Yaskawa INFORM job: DEMO_ROOF_SIDE_0625_3PAINT_34.JBI

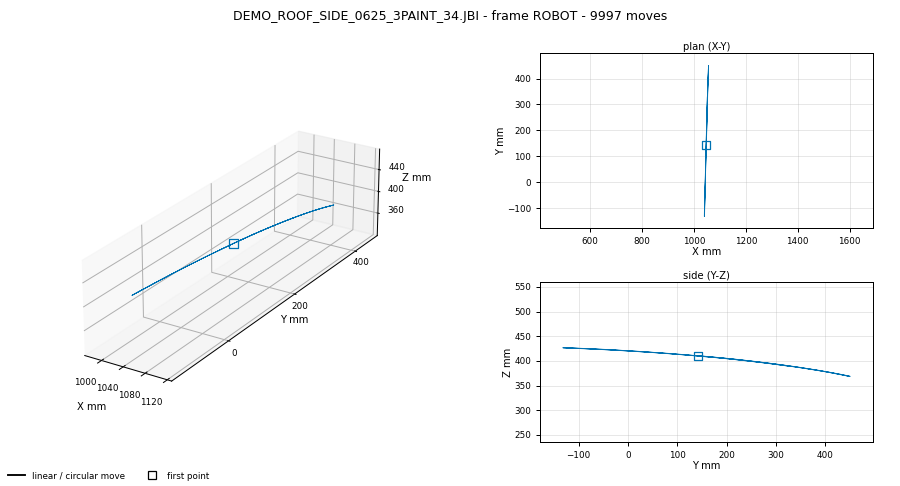
[picture p0: tool path of DEMO_ROOF_SIDE_0625_3PAINT_34.JBI in frame ROBOT, 9997 of 9997 moves have a stored position in this frame; points joined in program order, loops and branches not executed]
/JOB
//NAME DEMO_ROOF_SIDE_0625_3PAINT34
//POS
///NPOS 9997,0,0,0,0,0
///TOOL 0
///USER 0
///POSTYPE ROBOT
///RECTAN
///RCONF 1,0,0,0,0,0,0,0,0,0,0,0,0,0,0,0,0,0,0,0,0,0,0,0
C00000=1047.842,142.026,410.786,170.856,36.125,156.796
C00001=1047.849,142.311,410.761,170.858,36.127,156.797
C00002=1047.855,142.560,410.740,170.860,36.129,156.797
C00003=1047.861,142.809,410.718,170.862,36.131,156.797
C00004=1047.867,143.058,410.697,170.865,36.133,156.798
C00005=1047.873,143.307,410.675,170.866,36.135,156.798
C00006=1047.879,143.556,410.654,170.868,36.136,156.799
C00007=1047.886,143.805,410.633,170.870,36.138,156.799
C00008=1047.892,144.054,410.611,170.872,36.140,156.799
C00009=1047.898,144.303,410.590,170.874,36.142,156.800
C00010=1047.904,144.552,410.568,170.877,36.143,156.800
C00011=1047.910,144.801,410.546,170.878,36.145,156.800
C00012=1047.916,145.050,410.525,170.880,36.147,156.801
C00013=1047.922,145.299,410.504,170.882,36.149,156.801
C00014=1047.928,145.548,410.482,170.884,36.151,156.801
C00015=1047.934,145.797,410.460,170.887,36.153,156.802
C00016=1047.941,146.046,410.438,170.889,36.154,156.802
C00017=1047.947,146.295,410.416,170.890,36.156,156.802
C00018=1047.952,146.544,410.395,170.892,36.158,156.803
C00019=1047.959,146.793,410.373,170.894,36.160,156.803
C00020=1047.965,147.042,410.352,170.897,36.162,156.803
C00021=1047.971,147.291,410.330,170.899,36.164,156.804
C00022=1047.977,147.540,410.308,170.901,36.166,156.804
C00023=1047.983,147.788,410.287,170.903,36.167,156.804
C00024=1047.989,148.038,410.265,170.904,36.169,156.805
C00025=1047.995,148.287,410.243,170.907,36.171,156.805
C00026=1048.001,148.536,410.222,170.909,36.173,156.806
C00027=1048.007,148.785,410.199,170.911,36.175,156.806
C00028=1048.013,149.034,410.177,170.913,36.177,156.806
C00029=1048.019,149.283,410.156,170.915,36.179,156.807
C00030=1048.025,149.532,410.134,170.917,36.180,156.807
C00031=1048.032,149.780,410.112,170.919,36.182,156.807
C00032=1048.038,150.030,410.090,170.921,36.184,156.808
C00033=1048.043,150.279,410.068,170.923,36.186,156.808
C00034=1048.049,150.528,410.046,170.925,36.188,156.808
C00035=1048.055,150.776,410.024,170.927,36.190,156.809
C00036=1048.061,151.025,410.003,170.930,36.192,156.809
C00037=1048.067,151.275,409.981,170.931,36.193,156.809
C00038=1048.073,151.523,409.958,170.933,36.195,156.810
C00039=1048.079,151.773,409.936,170.935,36.197,156.810
C00040=1048.086,152.022,409.915,170.937,36.199,156.811
C00041=1048.092,152.270,409.892,170.940,36.201,156.811
C00042=1048.098,152.519,409.871,170.942,36.203,156.811
C00043=1048.103,152.768,409.848,170.944,36.205,156.812
C00044=1048.109,153.017,409.827,170.946,36.206,156.812
C00045=1048.116,153.266,409.805,170.947,36.208,156.812
C00046=1048.122,153.515,409.783,170.950,36.210,156.813
C00047=1048.128,153.764,409.760,170.952,36.212,156.813
C00048=1048.134,154.013,409.738,170.954,36.214,156.813
C00049=1048.140,154.262,409.716,170.956,36.216,156.814
C00050=1048.147,154.511,409.694,170.958,36.218,156.814
C00051=1048.152,154.760,409.672,170.961,36.219,156.815
C00052=1048.159,155.009,409.649,170.963,36.222,156.815
C00053=1048.164,155.257,409.628,170.965,36.224,156.815
C00054=1048.170,155.506,409.605,170.966,36.226,156.816
C00055=1048.176,155.755,409.584,170.968,36.227,156.816
C00056=1048.182,156.004,409.561,170.971,36.229,156.816
C00057=1048.188,156.254,409.539,170.973,36.231,156.817
C00058=1048.194,156.502,409.517,170.975,36.233,156.817
C00059=1048.201,156.751,409.495,170.977,36.235,156.818
C00060=1048.206,157.000,409.472,170.979,36.237,156.818
C00061=1048.212,157.249,409.450,170.982,36.239,156.818
C00062=1048.219,157.534,409.425,170.984,36.241,156.819
C00063=1048.226,157.820,409.399,170.986,36.244,156.819
C00064=1048.233,158.105,409.373,170.988,36.245,156.820
C00065=1048.240,158.390,409.348,170.991,36.248,156.820
C00066=1048.246,158.639,409.325,170.993,36.250,156.820
C00067=1048.252,158.888,409.304,170.995,36.252,156.821
C00068=1048.258,159.137,409.281,170.997,36.253,156.821
C00069=1048.265,159.386,409.259,170.999,36.255,156.821
C00070=1048.270,159.635,409.236,171.002,36.257,156.822
C00071=1048.277,159.884,409.214,171.004,36.259,156.822
C00072=1048.283,160.132,409.192,171.006,36.261,156.823
C00073=1048.288,160.382,409.169,171.008,36.263,156.823
C00074=1048.295,160.630,409.147,171.011,36.265,156.823
C00075=1048.301,160.879,409.124,171.013,36.267,156.824
C00076=1048.306,161.129,409.102,171.015,36.269,156.824
C00077=1048.312,161.378,409.079,171.017,36.271,156.825
C00078=1048.318,161.626,409.057,171.018,36.273,156.825
C00079=1048.324,161.875,409.034,171.021,36.275,156.825
C00080=1048.330,162.124,409.011,171.023,36.277,156.826
C00081=1048.335,162.373,408.988,171.025,36.279,156.826
C00082=1048.342,162.622,408.966,171.027,36.281,156.827
C00083=1048.347,162.871,408.943,171.030,36.283,156.827
C00084=1048.353,163.120,408.920,171.032,36.285,156.827
C00085=1048.359,163.369,408.897,171.034,36.287,156.828
C00086=1048.365,163.618,408.874,171.036,36.289,156.828
C00087=1048.371,163.866,408.852,171.038,36.292,156.829
C00088=1048.377,164.115,408.829,171.041,36.293,156.829
C00089=1048.382,164.364,408.806,171.043,36.295,156.829
C00090=1048.388,164.614,408.784,171.044,36.298,156.830
C00091=1048.394,164.862,408.761,171.046,36.300,156.830
C00092=1048.400,165.111,408.739,171.049,36.301,156.831
C00093=1048.406,165.360,408.716,171.051,36.304,156.831
C00094=1048.412,165.609,408.693,171.053,36.306,156.831
C00095=1048.417,165.858,408.670,171.055,36.308,156.832
C00096=1048.424,166.106,408.647,171.057,36.310,156.832
C00097=1048.429,166.355,408.624,171.060,36.312,156.833
C00098=1048.435,166.604,408.601,171.062,36.314,156.833
C00099=1048.441,166.853,408.579,171.064,36.316,156.833
C00100=1048.447,167.102,408.556,171.066,36.318,156.834
C00101=1048.452,167.351,408.533,171.069,36.320,156.834
C00102=1048.459,167.599,408.510,171.071,36.322,156.834
C00103=1048.465,167.849,408.487,171.073,36.324,156.835
C00104=1048.471,168.098,408.464,171.075,36.326,156.835
C00105=1048.477,168.347,408.441,171.077,36.328,156.836
C00106=1048.482,168.596,408.418,171.080,36.330,156.836
C00107=1048.489,168.844,408.395,171.082,36.332,156.837
C00108=1048.495,169.093,408.372,171.084,36.334,156.837
C00109=1048.501,169.341,408.349,171.086,36.336,156.837
C00110=1048.506,169.590,408.326,171.089,36.338,156.838
C00111=1048.512,169.839,408.303,171.091,36.340,156.838
C00112=1048.518,170.089,408.280,171.093,36.343,156.839
C00113=1048.525,170.337,408.258,171.095,36.344,156.839
C00114=1048.531,170.586,408.235,171.098,36.346,156.839
C00115=1048.536,170.835,408.212,171.100,36.349,156.840
C00116=1048.542,171.084,408.188,171.102,36.351,156.840
C00117=1048.548,171.332,408.165,171.104,36.352,156.841
C00118=1048.554,171.582,408.142,171.107,36.355,156.841
C00119=1048.561,171.831,408.119,171.109,36.357,156.841
C00120=1048.567,172.080,408.097,171.111,36.358,156.842
C00121=1048.573,172.328,408.073,171.113,36.361,156.842
C00122=1048.578,172.577,408.050,171.115,36.363,156.843
C00123=1048.585,172.826,408.027,171.118,36.365,156.843
C00124=1048.590,173.075,408.004,171.120,36.367,156.843
C00125=1048.596,173.323,407.980,171.122,36.369,156.844
C00126=1048.604,173.609,407.954,171.124,36.371,156.844
C00127=1048.610,173.893,407.928,171.127,36.374,156.845
C00128=1048.618,174.178,407.901,171.130,36.376,156.845
C00129=1048.624,174.463,407.875,171.132,36.378,156.846
C00130=1048.630,174.712,407.852,171.134,36.381,156.846
C00131=1048.636,174.961,407.828,171.137,36.382,156.846
C00132=1048.643,175.209,407.805,171.139,36.384,156.847
C00133=1048.649,175.458,407.782,171.141,36.387,156.847
C00134=1048.655,175.707,407.758,171.143,36.389,156.848
C00135=1048.661,175.956,407.735,171.146,36.390,156.848
C00136=1048.667,176.205,407.712,171.148,36.393,156.849
C00137=1048.673,176.453,407.689,171.150,36.395,156.849
C00138=1048.679,176.703,407.665,171.152,36.397,156.849
C00139=1048.685,176.951,407.642,171.155,36.399,156.850
C00140=1048.691,177.200,407.619,171.158,36.401,156.850
C00141=1048.698,177.449,407.596,171.160,36.403,156.851
C00142=1048.704,177.697,407.572,171.162,36.405,156.851
C00143=1048.710,177.946,407.550,171.164,36.407,156.851
C00144=1048.716,178.195,407.525,171.167,36.409,156.852
C00145=1048.722,178.444,407.503,171.169,36.411,156.852
C00146=1048.728,178.692,407.479,171.171,36.413,156.853
C00147=1048.734,178.942,407.456,171.173,36.415,156.853
C00148=1048.740,179.191,407.433,171.176,36.417,156.853
C00149=1048.746,179.439,407.409,171.178,36.420,156.854
C00150=1048.753,179.689,407.386,171.180,36.422,156.854
C00151=1048.759,179.937,407.362,171.182,36.423,156.855
C00152=1048.765,180.187,407.339,171.186,36.426,156.855
C00153=1048.772,180.435,407.316,171.188,36.428,156.855
C00154=1048.778,180.683,407.292,171.190,36.429,156.856
C00155=1048.784,180.933,407.269,171.192,36.432,156.856
C00156=1048.790,181.181,407.245,171.195,36.434,156.857
C00157=1048.796,181.430,407.222,171.197,36.436,156.857
C00158=1048.802,181.679,407.198,171.199,36.438,156.858
C00159=1048.808,181.928,407.175,171.201,36.440,156.858
C00160=1048.815,182.177,407.151,171.204,36.442,156.858
C00161=1048.821,182.425,407.127,171.207,36.444,156.859
C00162=1048.827,182.674,407.104,171.209,36.447,156.859
C00163=1048.833,182.923,407.080,171.211,36.448,156.860
C00164=1048.840,183.172,407.057,171.213,36.450,156.860
C00165=1048.846,183.421,407.033,171.216,36.453,156.860
C00166=1048.852,183.670,407.009,171.218,36.454,156.861
C00167=1048.858,183.918,406.986,171.220,36.456,156.861
C00168=1048.865,184.167,406.962,171.222,36.459,156.862
C00169=1048.871,184.416,406.939,171.226,36.461,156.862
C00170=1048.876,184.664,406.915,171.228,36.463,156.863
C00171=1048.882,184.914,406.891,171.230,36.465,156.863
C00172=1048.888,185.163,406.867,171.233,36.468,156.864
C00173=1048.894,185.411,406.843,171.235,36.470,156.864
C00174=1048.900,185.660,406.819,171.237,36.472,156.864
C00175=1048.906,185.908,406.795,171.239,36.475,156.865
C00176=1048.911,186.157,406.771,171.242,36.477,156.865
C00177=1048.917,186.406,406.747,171.244,36.479,156.866
C00178=1048.922,186.655,406.723,171.246,36.481,156.866
C00179=1048.929,186.904,406.699,171.249,36.484,156.867
C00180=1048.934,187.153,406.675,171.252,36.486,156.867
C00181=1048.940,187.401,406.651,171.254,36.488,156.868
C00182=1048.947,187.650,406.627,171.256,36.490,156.868
C00183=1048.952,187.899,406.603,171.259,36.493,156.869
C00184=1048.959,188.148,406.579,171.261,36.495,156.869
C00185=1048.964,188.396,406.555,171.263,36.497,156.869
C00186=1048.971,188.645,406.531,171.265,36.500,156.870
C00187=1048.976,188.894,406.506,171.269,36.501,156.870
C00188=1048.983,189.143,406.482,171.271,36.504,156.871
C00189=1048.988,189.391,406.458,171.273,36.506,156.871
C00190=1048.995,189.676,406.431,171.275,36.509,156.872
C00191=1049.002,189.960,406.403,171.279,36.511,156.872
C00192=1049.009,190.244,406.376,171.281,36.514,156.873
C00193=1049.016,190.529,406.347,171.284,36.517,156.873
C00194=1049.022,190.777,406.323,171.287,36.519,156.874
C00195=1049.028,191.027,406.299,171.289,36.521,156.874
C00196=1049.034,191.275,406.275,171.291,36.523,156.875
C00197=1049.040,191.524,406.250,171.293,36.526,156.875
C00198=1049.046,191.772,406.227,171.296,36.528,156.876
C00199=1049.051,192.022,406.202,171.299,36.531,156.876
C00200=1049.058,192.270,406.178,171.301,36.532,156.877
C00201=1049.063,192.519,406.154,171.304,36.535,156.877
C00202=1049.069,192.768,406.130,171.306,36.537,156.878
C00203=1049.076,193.016,406.105,171.308,36.540,156.878
C00204=1049.082,193.264,406.081,171.311,36.541,156.878
C00205=1049.088,193.514,406.057,171.314,36.544,156.879
C00206=1049.094,193.763,406.033,171.316,36.546,156.879
C00207=1049.100,194.011,406.008,171.318,36.549,156.880
C00208=1049.105,194.261,405.984,171.321,36.551,156.880
C00209=1049.112,194.508,405.959,171.324,36.553,156.881
C00210=1049.118,194.758,405.935,171.326,36.555,156.881
C00211=1049.124,195.007,405.911,171.328,36.558,156.882
C00212=1049.130,195.255,405.886,171.331,36.560,156.882
C00213=1049.137,195.503,405.862,171.333,36.562,156.883
C00214=1049.142,195.752,405.837,171.336,36.564,156.883
C00215=1049.149,196.001,405.813,171.339,36.567,156.884
C00216=1049.154,196.250,405.789,171.341,36.569,156.884
C00217=1049.160,196.498,405.764,171.343,36.572,156.885
C00218=1049.167,196.747,405.740,171.346,36.574,156.885
C00219=1049.173,196.997,405.715,171.349,36.576,156.885
C00220=1049.179,197.244,405.691,171.351,36.578,156.886
C00221=1049.185,197.494,405.666,171.353,36.581,156.886
C00222=1049.191,197.743,405.642,171.357,36.583,156.887
C00223=1049.197,197.990,405.617,171.359,36.585,156.887
C00224=1049.203,198.240,405.593,171.361,36.587,156.888
C00225=1049.210,198.488,405.568,171.363,36.590,156.888
C00226=1049.216,198.737,405.543,171.367,36.592,156.889
C00227=1049.222,198.986,405.519,171.369,36.595,156.889
C00228=1049.228,199.234,405.494,171.371,36.597,156.890
C00229=1049.235,199.483,405.470,171.373,36.599,156.890
C00230=1049.241,199.732,405.445,171.377,36.601,156.891
C00231=1049.246,199.981,405.421,171.379,36.604,156.891
C00232=1049.253,200.229,405.396,171.381,36.606,156.892
C00233=1049.259,200.478,405.371,171.384,36.609,156.892
C00234=1049.266,200.727,405.347,171.387,36.611,156.893
C00235=1049.271,200.975,405.322,171.389,36.613,156.893
C00236=1049.277,201.224,405.298,171.392,36.615,156.893
C00237=1049.284,201.473,405.273,171.395,36.618,156.894
C00238=1049.290,201.721,405.247,171.397,36.620,156.894
C00239=1049.296,201.970,405.223,171.399,36.623,156.895
C00240=1049.302,202.219,405.198,171.402,36.625,156.895
C00241=1049.308,202.468,405.173,171.405,36.627,156.896
C00242=1049.314,202.717,405.148,171.407,36.630,156.896
C00243=1049.320,202.965,405.123,171.410,36.632,156.897
C00244=1049.325,203.214,405.098,171.412,36.635,156.897
C00245=1049.332,203.463,405.073,171.415,36.638,156.898
C00246=1049.339,203.711,405.048,171.418,36.640,156.898
C00247=1049.344,203.960,405.024,171.420,36.642,156.899
C00248=1049.350,204.208,404.999,171.423,36.645,156.899
C00249=1049.356,204.457,404.973,171.426,36.647,156.900
C00250=1049.362,204.706,404.949,171.428,36.650,156.900
C00251=1049.368,204.955,404.923,171.430,36.652,156.901
C00252=1049.374,205.203,404.898,171.433,36.655,156.901
C00253=1049.380,205.452,404.873,171.436,36.657,156.902
C00254=1049.406,206.504,404.768,171.671,36.754,156.922
C00255=1049.413,206.762,404.740,171.673,36.758,156.923
C00256=1049.420,207.019,404.713,171.674,36.761,156.924
C00257=1049.426,207.278,404.686,171.677,36.764,156.925
C00258=1049.433,207.535,404.659,171.678,36.768,156.925
C00259=1049.440,207.783,404.633,171.681,36.771,156.926
C00260=1049.446,208.032,404.606,171.683,36.774,156.927
C00261=1049.452,208.281,404.581,171.685,36.777,156.927
C00262=1049.459,208.529,404.555,171.687,36.781,156.928
C00263=1049.465,208.778,404.528,171.689,36.784,156.929
C00264=1049.472,209.026,404.502,171.691,36.787,156.929
C00265=1049.478,209.275,404.476,171.693,36.791,156.930
C00266=1049.485,209.523,404.450,171.695,36.794,156.931
C00267=1049.491,209.772,404.423,171.697,36.797,156.931
C00268=1049.498,210.020,404.397,171.699,36.800,156.932
C00269=1049.504,210.269,404.370,171.701,36.804,156.933
C00270=1049.511,210.518,404.344,171.703,36.807,156.933
C00271=1049.517,210.766,404.318,171.705,36.810,156.934
C00272=1049.523,211.015,404.292,171.707,36.813,156.935
C00273=1049.530,211.263,404.265,171.709,36.816,156.935
C00274=1049.536,211.511,404.239,171.711,36.820,156.936
C00275=1049.543,211.760,404.212,171.714,36.823,156.937
C00276=1049.549,212.008,404.186,171.715,36.826,156.937
C00277=1049.556,212.258,404.159,171.718,36.829,156.938
C00278=1049.562,212.506,404.133,171.719,36.832,156.939
C00279=1049.568,212.754,404.106,171.721,36.836,156.940
C00280=1049.575,213.003,404.080,171.724,36.839,156.940
C00281=1049.581,213.251,404.053,171.725,36.843,156.941
C00282=1049.588,213.500,404.027,171.728,36.846,156.942
C00283=1049.594,213.748,404.000,171.729,36.849,156.942
C00284=1049.599,213.996,403.974,171.732,36.852,156.943
C00285=1049.606,214.245,403.947,171.734,36.856,156.944
C00286=1049.612,214.494,403.921,171.736,36.859,156.944
C00287=1049.619,214.742,403.894,171.738,36.862,156.945
C00288=1049.625,214.991,403.867,171.740,36.865,156.946
C00289=1049.632,215.239,403.841,171.742,36.868,156.946
C00290=1049.638,215.488,403.814,171.744,36.872,156.947
C00291=1049.645,215.737,403.788,171.747,36.875,156.948
C00292=1049.651,215.985,403.761,171.748,36.878,156.948
C00293=1049.658,216.233,403.734,171.751,36.881,156.949
C00294=1049.664,216.481,403.708,171.753,36.884,156.950
C00295=1049.670,216.730,403.681,171.755,36.888,156.951
C00296=1049.677,216.979,403.655,171.757,36.891,156.951
C00297=1049.683,217.228,403.627,171.759,36.894,156.952
C00298=1049.690,217.476,403.601,171.761,36.898,156.953
C00299=1049.696,217.725,403.574,171.763,36.901,156.953
C00300=1049.702,217.972,403.547,171.766,36.904,156.954
C00301=1049.709,218.221,403.521,171.767,36.907,156.955
C00302=1049.716,218.470,403.494,171.770,36.910,156.955
C00303=1049.722,218.718,403.468,171.772,36.913,156.956
C00304=1049.729,218.967,403.440,171.774,36.917,156.957
C00305=1049.735,219.215,403.413,171.776,36.920,156.957
C00306=1049.742,219.464,403.387,171.778,36.923,156.958
C00307=1049.748,219.712,403.360,171.780,36.926,156.959
C00308=1049.755,219.960,403.333,171.782,36.929,156.959
C00309=1049.761,220.209,403.306,171.785,36.932,156.960
C00310=1049.767,220.458,403.279,171.787,36.936,156.961
C00311=1049.774,220.721,403.251,171.789,36.939,156.961
C00312=1049.781,220.984,403.222,171.791,36.942,156.962
C00313=1049.788,221.248,403.194,171.794,36.946,156.963
C00314=1049.795,221.511,403.165,171.796,36.949,156.963
C00315=1049.801,221.759,403.138,171.799,36.952,156.964
C00316=1049.807,222.008,403.111,171.800,36.955,156.965
C00317=1049.814,222.256,403.083,171.802,36.959,156.966
C00318=1049.820,222.505,403.057,171.805,36.962,156.966
C00319=1049.827,222.753,403.030,171.806,36.966,156.967
C00320=1049.833,223.001,403.003,171.809,36.969,156.968
C00321=1049.839,223.250,402.976,171.811,36.972,156.968
C00322=1049.846,223.499,402.948,171.814,36.975,156.969
C00323=1049.852,223.747,402.921,171.815,36.978,156.970
C00324=1049.858,223.996,402.894,171.818,36.981,156.970
C00325=1049.864,224.244,402.867,171.820,36.985,156.971
C00326=1049.872,224.492,402.840,171.822,36.988,156.972
C00327=1049.878,224.741,402.813,171.824,36.991,156.972
C00328=1049.884,224.989,402.786,171.826,36.994,156.973
C00329=1049.890,225.238,402.759,171.829,36.997,156.974
C00330=1049.897,225.486,402.731,171.831,37.001,156.974
C00331=1049.903,225.734,402.703,171.833,37.004,156.975
C00332=1049.910,225.983,402.676,171.835,37.007,156.976
C00333=1049.916,226.232,402.649,171.838,37.010,156.976
C00334=1049.923,226.480,402.623,171.840,37.013,156.977
C00335=1049.929,226.728,402.595,171.843,37.016,156.978
C00336=1049.936,226.977,402.568,171.844,37.019,156.978
C00337=1049.942,227.226,402.540,171.846,37.023,156.979
C00338=1049.949,227.473,402.513,171.849,37.026,156.980
C00339=1049.955,227.722,402.486,171.851,37.029,156.980
C00340=1049.962,227.971,402.458,171.853,37.032,156.981
C00341=1049.968,228.219,402.431,171.855,37.035,156.982
C00342=1049.974,228.468,402.404,171.858,37.038,156.982
C00343=1049.981,228.716,402.376,171.860,37.042,156.983
C00344=1049.988,228.964,402.349,171.863,37.045,156.984
C00345=1049.994,229.213,402.322,171.865,37.048,156.984
C00346=1050.000,229.461,402.294,171.867,37.051,156.985
C00347=1050.007,229.710,402.266,171.869,37.054,156.986
C00348=1050.013,229.958,402.238,171.871,37.057,156.986
C00349=1050.019,230.206,402.211,171.874,37.061,156.987
C00350=1050.026,230.455,402.184,171.876,37.064,156.988
C00351=1050.032,230.703,402.156,171.878,37.067,156.988
C00352=1050.039,230.952,402.129,171.880,37.070,156.989
C00353=1050.045,231.200,402.101,171.883,37.073,156.990
C00354=1050.052,231.448,402.073,171.885,37.076,156.990
C00355=1050.057,231.697,402.046,171.888,37.080,156.991
C00356=1050.064,231.946,402.018,171.889,37.083,156.992
C00357=1050.070,232.194,401.991,171.892,37.086,156.993
C00358=1050.077,232.442,401.963,171.894,37.089,156.993
C00359=1050.084,232.690,401.935,171.896,37.092,156.994
C00360=1050.090,232.939,401.908,171.899,37.095,156.995
C00361=1050.096,233.188,401.879,171.901,37.099,156.995
C00362=1050.102,233.435,401.852,171.904,37.102,156.996
C00363=1050.109,233.684,401.824,171.905,37.105,156.997
C00364=1050.116,233.932,401.796,171.908,37.108,156.997
C00365=1050.122,234.181,401.768,171.910,37.111,156.998
C00366=1050.128,234.429,401.741,171.913,37.115,156.999
C00367=1050.135,234.685,401.712,171.915,37.118,156.999
C00368=1050.141,234.940,401.683,171.918,37.121,157.000
C00369=1050.148,235.197,401.655,171.920,37.124,157.001
C00370=1050.154,235.452,401.626,171.923,37.128,157.002
C00371=1050.160,235.700,401.598,171.924,37.131,157.002
C00372=1050.167,235.949,401.571,171.927,37.133,157.003
C00373=1050.174,236.197,401.543,171.929,37.137,157.004
C00374=1050.180,236.446,401.515,171.932,37.140,157.004
C00375=1050.186,236.695,401.487,171.934,37.143,157.005
C00376=1050.193,236.942,401.459,171.937,37.146,157.006
C00377=1050.199,237.190,401.430,171.939,37.149,157.006
C00378=1050.205,237.439,401.403,171.941,37.152,157.007
C00379=1050.212,237.687,401.375,171.944,37.155,157.008
C00380=1050.219,237.936,401.347,171.945,37.159,157.008
C00381=1050.225,238.184,401.319,171.948,37.162,157.009
C00382=1050.231,238.433,401.291,171.950,37.165,157.010
C00383=1050.238,238.681,401.263,171.953,37.168,157.010
C00384=1050.244,238.930,401.234,171.955,37.171,157.011
C00385=1050.251,239.178,401.207,171.958,37.174,157.012
C00386=1050.257,239.426,401.179,171.960,37.178,157.012
C00387=1050.263,239.674,401.151,171.963,37.181,157.013
C00388=1050.270,239.922,401.123,171.965,37.184,157.014
C00389=1050.276,240.171,401.094,171.968,37.187,157.015
C00390=1050.283,240.419,401.066,171.970,37.190,157.015
C00391=1050.290,240.667,401.038,171.973,37.193,157.016
C00392=1050.296,240.916,401.010,171.975,37.196,157.016
C00393=1050.302,241.164,400.982,171.977,37.200,157.017
C00394=1050.309,241.413,400.954,171.980,37.203,157.018
C00395=1050.315,241.661,400.925,171.981,37.206,157.018
C00396=1050.322,241.909,400.897,171.984,37.209,157.019
C00397=1050.328,242.158,400.868,171.986,37.212,157.020
C00398=1050.334,242.406,400.840,171.989,37.215,157.021
C00399=1050.341,242.655,400.812,171.991,37.219,157.021
C00400=1050.347,242.903,400.783,171.994,37.221,157.022
C00401=1050.354,243.151,400.756,171.996,37.225,157.023
C00402=1050.360,243.400,400.727,171.999,37.228,157.023
C00403=1050.366,243.648,400.698,172.001,37.231,157.024
C00404=1050.373,243.896,400.670,172.004,37.234,157.025
C00405=1050.379,244.145,400.641,172.006,37.237,157.025
C00406=1050.386,244.393,400.613,172.009,37.240,157.026
C00407=1050.392,244.641,400.585,172.011,37.244,157.027
C00408=1050.398,244.890,400.556,172.014,37.247,157.027
C00409=1050.405,245.138,400.528,172.016,37.250,157.028
C00410=1050.411,245.386,400.499,172.019,37.253,157.029
C00411=1050.418,245.635,400.471,172.021,37.256,157.030
C00412=1050.424,245.883,400.442,172.024,37.260,157.030
C00413=1050.430,246.131,400.413,172.026,37.263,157.031
C00414=1050.436,246.380,400.385,172.029,37.266,157.032
C00415=1050.442,246.628,400.356,172.031,37.269,157.032
C00416=1050.449,246.876,400.328,172.034,37.272,157.033
C00417=1050.455,247.124,400.299,172.036,37.276,157.034
C00418=1050.462,247.372,400.270,172.039,37.279,157.034
C00419=1050.468,247.621,400.241,172.041,37.282,157.035
C00420=1050.474,247.869,400.213,172.044,37.285,157.036
C00421=1050.480,248.117,400.184,172.046,37.288,157.036
C00422=1050.486,248.366,400.154,172.049,37.291,157.037
C00423=1050.493,248.615,400.126,172.051,37.294,157.038
C00424=1050.499,248.865,400.097,172.054,37.298,157.039
C00425=1050.505,249.115,400.069,172.056,37.301,157.039
C00426=1050.512,249.365,400.039,172.059,37.304,157.040
C00427=1050.518,249.613,400.010,172.061,37.307,157.041
C00428=1050.524,249.861,399.981,172.064,37.311,157.042
C00429=1050.531,250.109,399.952,172.066,37.314,157.042
C00430=1050.537,250.358,399.923,172.069,37.317,157.043
C00431=1050.543,250.606,399.895,172.071,37.320,157.044
C00432=1050.549,250.855,399.866,172.074,37.323,157.044
C00433=1050.555,251.103,399.837,172.076,37.327,157.045
C00434=1050.562,251.350,399.808,172.079,37.330,157.046
C00435=1050.569,251.599,399.779,172.081,37.333,157.046
C00436=1050.575,251.847,399.750,172.084,37.336,157.047
C00437=1050.582,252.096,399.721,172.086,37.339,157.048
C00438=1050.588,252.344,399.692,172.089,37.343,157.048
C00439=1050.594,252.592,399.663,172.091,37.345,157.049
C00440=1050.600,252.840,399.634,172.094,37.348,157.050
C00441=1050.606,253.089,399.606,172.097,37.352,157.051
C00442=1050.613,253.338,399.576,172.100,37.355,157.051
C00443=1050.620,253.585,399.548,172.102,37.358,157.052
C00444=1050.626,253.833,399.519,172.105,37.361,157.053
C00445=1050.633,254.082,399.490,172.107,37.364,157.053
C00446=1050.639,254.330,399.461,172.110,37.368,157.054
C00447=1050.646,254.579,399.431,172.112,37.371,157.055
C00448=1050.652,254.827,399.402,172.114,37.374,157.055
C00449=1050.659,255.074,399.372,172.117,37.377,157.056
C00450=1050.665,255.322,399.343,172.120,37.380,157.057
C00451=1050.671,255.570,399.314,172.123,37.383,157.057
C00452=1050.678,255.819,399.285,172.126,37.386,157.058
C00453=1050.684,256.067,399.256,172.128,37.389,157.059
C00454=1050.690,256.316,399.227,172.130,37.392,157.060
C00455=1050.697,256.564,399.198,172.133,37.396,157.060
C00456=1050.704,256.812,399.169,172.136,37.399,157.061
C00457=1050.711,257.060,399.140,172.138,37.402,157.062
C00458=1050.717,257.308,399.110,172.142,37.405,157.062
C00459=1050.724,257.557,399.081,172.144,37.408,157.063
C00460=1050.730,257.805,399.052,172.147,37.412,157.064
C00461=1050.736,258.053,399.023,172.149,37.414,157.064
C00462=1050.743,258.301,398.994,172.152,37.417,157.065
C00463=1050.750,258.549,398.963,172.154,37.421,157.066
C00464=1050.756,258.797,398.934,172.157,37.424,157.067
C00465=1050.762,259.046,398.905,172.160,37.427,157.067
C00466=1050.769,259.294,398.876,172.163,37.430,157.068
C00467=1050.776,259.542,398.846,172.165,37.433,157.069
C00468=1050.782,259.790,398.817,172.168,37.436,157.069
C00469=1050.789,260.039,398.788,172.170,37.440,157.070
C00470=1050.795,260.287,398.759,172.173,37.443,157.071
C00471=1050.802,260.535,398.729,172.176,37.445,157.071
C00472=1050.809,260.783,398.700,172.179,37.449,157.072
C00473=1050.815,261.032,398.671,172.181,37.452,157.073
C00474=1050.822,261.280,398.640,172.184,37.455,157.073
C00475=1050.828,261.528,398.611,172.186,37.458,157.074
C00476=1050.834,261.776,398.582,172.190,37.461,157.075
C00477=1050.842,262.024,398.552,172.192,37.464,157.076
C00478=1050.848,262.272,398.523,172.195,37.467,157.076
C00479=1050.855,262.521,398.493,172.197,37.470,157.077
C00480=1050.861,262.769,398.464,172.201,37.473,157.078
C00481=1050.868,263.018,398.435,172.203,37.477,157.078
C00482=1050.874,263.265,398.404,172.206,37.480,157.079
C00483=1050.880,263.513,398.374,172.208,37.483,157.080
C00484=1050.887,263.762,398.345,172.211,37.486,157.080
C00485=1050.894,264.009,398.315,172.214,37.489,157.081
C00486=1050.899,264.258,398.286,172.217,37.493,157.082
C00487=1050.907,264.506,398.256,172.219,37.495,157.083
C00488=1050.913,264.754,398.227,172.222,37.499,157.083
C00489=1050.919,265.002,398.196,172.224,37.502,157.084
C00490=1050.926,265.250,398.166,172.228,37.505,157.085
C00491=1050.932,265.498,398.137,172.230,37.508,157.085
C00492=1050.938,265.747,398.106,172.233,37.512,157.086
C00493=1050.945,265.994,398.077,172.235,37.515,157.087
C00494=1050.951,266.243,398.047,172.239,37.518,157.088
C00495=1050.958,266.491,398.017,172.242,37.521,157.088
C00496=1050.965,266.739,397.987,172.244,37.525,157.089
C00497=1050.970,266.987,397.957,172.247,37.527,157.090
C00498=1050.978,267.236,397.927,172.250,37.531,157.091
C00499=1050.984,267.483,397.897,172.253,37.534,157.091
C00500=1050.990,267.731,397.867,172.255,37.537,157.092
C00501=1050.997,267.980,397.837,172.258,37.540,157.093
C00502=1051.003,268.228,397.807,172.261,37.544,157.093
C00503=1051.010,268.476,397.777,172.264,37.547,157.094
C00504=1051.016,268.723,397.747,172.266,37.550,157.095
C00505=1051.023,268.972,397.716,172.269,37.553,157.096
C00506=1051.029,269.220,397.687,172.272,37.556,157.096
C00507=1051.035,269.469,397.657,172.275,37.559,157.097
C00508=1051.042,269.716,397.627,172.278,37.563,157.098
C00509=1051.048,269.965,397.596,172.281,37.566,157.098
C00510=1051.055,270.212,397.566,172.284,37.569,157.099
C00511=1051.061,270.461,397.536,172.286,37.572,157.100
C00512=1051.068,270.708,397.506,172.289,37.576,157.101
C00513=1051.074,270.957,397.475,172.292,37.579,157.101
C00514=1051.080,271.205,397.445,172.295,37.582,157.102
C00515=1051.087,271.453,397.415,172.297,37.585,157.103
C00516=1051.094,271.701,397.384,172.301,37.588,157.104
C00517=1051.100,271.949,397.354,172.303,37.591,157.104
C00518=1051.107,272.197,397.324,172.306,37.595,157.105
C00519=1051.113,272.445,397.294,172.309,37.598,157.106
C00520=1051.120,272.693,397.263,172.312,37.601,157.106
C00521=1051.125,272.941,397.233,172.315,37.605,157.107
C00522=1051.133,273.189,397.203,172.318,37.607,157.108
C00523=1051.138,273.437,397.172,172.321,37.611,157.109
C00524=1051.145,273.686,397.142,172.323,37.614,157.109
C00525=1051.152,273.934,397.111,172.327,37.617,157.110
C00526=1051.158,274.181,397.080,172.329,37.621,157.111
C00527=1051.165,274.430,397.050,172.332,37.624,157.112
C00528=1051.171,274.677,397.020,172.335,37.627,157.112
C00529=1051.177,274.926,396.989,172.338,37.630,157.113
C00530=1051.184,275.174,396.959,172.341,37.634,157.114
C00531=1051.190,275.422,396.929,172.344,37.636,157.114
C00532=1051.197,275.670,396.897,172.347,37.640,157.115
C00533=1051.203,275.917,396.867,172.349,37.643,157.116
C00534=1051.209,276.166,396.836,172.353,37.646,157.117
C00535=1051.216,276.418,396.805,172.355,37.650,157.117
C00536=1051.222,276.671,396.774,172.359,37.653,157.118
C00537=1051.229,276.923,396.743,172.361,37.656,157.119
C00538=1051.237,277.176,396.711,172.364,37.659,157.120
C00539=1051.243,277.424,396.681,172.368,37.663,157.121
C00540=1051.249,277.672,396.650,172.370,37.666,157.121
C00541=1051.256,277.920,396.619,172.374,37.669,157.122
C00542=1051.262,278.168,396.589,172.376,37.673,157.123
C00543=1051.269,278.416,396.558,172.379,37.676,157.123
C00544=1051.275,278.664,396.527,172.382,37.679,157.124
C00545=1051.281,278.912,396.497,172.385,37.683,157.125
C00546=1051.288,279.160,396.465,172.389,37.685,157.126
C00547=1051.294,279.408,396.434,172.391,37.689,157.126
C00548=1051.301,279.655,396.404,172.394,37.692,157.127
C00549=1051.308,279.904,396.373,172.397,37.695,157.128
C00550=1051.314,280.152,396.342,172.400,37.699,157.129
C00551=1051.321,280.400,396.311,172.403,37.702,157.130
C00552=1051.327,280.647,396.280,172.406,37.705,157.130
C00553=1051.333,280.896,396.249,172.409,37.708,157.131
C00554=1051.340,281.144,396.218,172.412,37.712,157.132
C00555=1051.346,281.391,396.187,172.415,37.715,157.133
C00556=1051.353,281.640,396.156,172.418,37.718,157.133
C00557=1051.359,281.887,396.125,172.421,37.722,157.134
C00558=1051.366,282.135,396.093,172.424,37.725,157.135
C00559=1051.372,282.383,396.063,172.427,37.729,157.136
C00560=1051.379,282.631,396.031,172.430,37.732,157.136
C00561=1051.384,282.880,396.000,172.433,37.735,157.137
C00562=1051.391,283.128,395.969,172.436,37.738,157.138
C00563=1051.397,283.375,395.938,172.439,37.742,157.139
C00564=1051.404,283.623,395.906,172.442,37.745,157.139
C00565=1051.410,283.871,395.876,172.446,37.748,157.140
C00566=1051.417,284.119,395.844,172.448,37.752,157.141
C00567=1051.424,284.367,395.813,172.452,37.755,157.142
C00568=1051.430,284.615,395.781,172.454,37.758,157.142
C00569=1051.436,284.863,395.751,172.458,37.761,157.143
C00570=1051.443,285.111,395.719,172.461,37.765,157.144
C00571=1051.450,285.359,395.688,172.464,37.768,157.145
C00572=1051.456,285.607,395.657,172.467,37.771,157.145
C00573=1051.463,285.855,395.625,172.470,37.775,157.146
C00574=1051.470,286.103,395.594,172.473,37.778,157.147
C00575=1051.476,286.350,395.563,172.477,37.781,157.148
C00576=1051.482,286.598,395.532,172.479,37.784,157.149
C00577=1051.489,286.846,395.500,172.483,37.788,157.149
C00578=1051.496,287.094,395.469,172.485,37.791,157.150
C00579=1051.503,287.342,395.438,172.489,37.795,157.151
C00580=1051.509,287.590,395.406,172.491,37.798,157.152
C00581=1051.515,287.838,395.374,172.495,37.801,157.152
C00582=1051.522,288.086,395.343,172.498,37.804,157.153
C00583=1051.529,288.334,395.311,172.501,37.808,157.154
C00584=1051.535,288.582,395.280,172.504,37.811,157.155
C00585=1051.541,288.830,395.248,172.507,37.815,157.156
C00586=1051.548,289.077,395.217,172.510,37.818,157.156
C00587=1051.554,289.325,395.185,172.514,37.821,157.157
C00588=1051.561,289.573,395.154,172.516,37.824,157.158
C00589=1051.567,289.821,395.122,172.520,37.828,157.159
C00590=1051.574,290.069,395.090,172.523,37.831,157.159
C00591=1051.581,290.333,395.056,172.526,37.835,157.160
C00592=1051.588,290.597,395.023,172.530,37.838,157.161
C00593=1051.594,290.861,394.989,172.533,37.842,157.162
C00594=1051.602,291.125,394.955,172.536,37.846,157.163
C00595=1051.609,291.373,394.924,172.540,37.849,157.164
C00596=1051.615,291.620,394.891,172.542,37.852,157.164
C00597=1051.622,291.868,394.860,172.546,37.856,157.165
C00598=1051.628,292.116,394.828,172.550,37.859,157.166
C00599=1051.634,292.364,394.796,172.552,37.863,157.167
C00600=1051.641,292.611,394.764,172.556,37.866,157.168
C00601=1051.648,292.860,394.732,172.559,37.870,157.168
C00602=1051.654,293.108,394.700,172.562,37.872,157.169
C00603=1051.661,293.355,394.668,172.566,37.876,157.170
C00604=1051.667,293.603,394.636,172.568,37.879,157.171
C00605=1051.674,293.851,394.605,172.572,37.883,157.171
C00606=1051.681,294.098,394.573,172.575,37.886,157.172
C00607=1051.687,294.347,394.541,172.578,37.890,157.173
C00608=1051.694,294.595,394.509,172.582,37.893,157.174
C00609=1051.700,294.842,394.476,172.584,37.896,157.175
C00610=1051.707,295.090,394.445,172.588,37.900,157.176
C00611=1051.713,295.338,394.412,172.591,37.903,157.176
C00612=1051.720,295.586,394.381,172.594,37.907,157.177
C00613=1051.726,295.833,394.348,172.598,37.910,157.178
C00614=1051.733,296.081,394.317,172.601,37.914,157.179
C00615=1051.739,296.329,394.284,172.604,37.917,157.180
C00616=1051.746,296.577,394.253,172.608,37.920,157.180
C00617=1051.752,296.824,394.220,172.611,37.924,157.181
C00618=1051.758,297.072,394.187,172.614,37.928,157.182
C00619=1051.764,297.320,394.155,172.617,37.931,157.183
C00620=1051.771,297.567,394.123,172.621,37.935,157.184
C00621=1051.778,297.816,394.090,172.624,37.938,157.185
C00622=1051.784,298.064,394.058,172.627,37.942,157.185
C00623=1051.790,298.311,394.025,172.631,37.945,157.186
C00624=1051.797,298.559,393.992,172.634,37.949,157.187
C00625=1051.804,298.807,393.961,172.637,37.952,157.188
C00626=1051.810,299.054,393.928,172.640,37.956,157.189
C00627=1051.816,299.302,393.895,172.643,37.960,157.190
C00628=1051.822,299.550,393.863,172.647,37.963,157.190
C00629=1051.828,299.798,393.831,172.651,37.966,157.191
C00630=1051.835,300.045,393.798,172.653,37.970,157.192
C00631=1051.842,300.293,393.765,172.657,37.973,157.193
C00632=1051.849,300.541,393.733,172.661,37.977,157.194
C00633=1051.855,300.789,393.700,172.664,37.981,157.195
C00634=1051.861,301.036,393.667,172.667,37.984,157.195
C00635=1051.868,301.284,393.636,172.671,37.987,157.196
C00636=1051.874,301.532,393.603,172.674,37.991,157.197
C00637=1051.881,301.780,393.570,172.677,37.995,157.198
C00638=1051.887,302.028,393.537,172.681,37.998,157.199
C00639=1051.894,302.275,393.504,172.684,38.002,157.200
C00640=1051.900,302.523,393.472,172.687,38.005,157.200
C00641=1051.907,302.770,393.439,172.691,38.009,157.201
C00642=1051.914,303.018,393.406,172.694,38.012,157.202
C00643=1051.920,303.266,393.374,172.698,38.016,157.203
C00644=1051.926,303.514,393.341,172.701,38.019,157.204
C00645=1051.933,303.761,393.308,172.704,38.023,157.205
C00646=1051.940,304.009,393.275,172.708,38.027,157.206
C00647=1051.947,304.289,393.238,172.712,38.031,157.206
C00648=1051.955,304.568,393.201,172.715,38.035,157.207
C00649=1051.963,304.849,393.164,172.719,38.039,157.208
C00650=1051.970,305.129,393.127,172.723,38.042,157.209
C00651=1051.976,305.376,393.094,172.727,38.046,157.210
C00652=1051.983,305.624,393.061,172.730,38.050,157.211
C00653=1051.989,305.872,393.028,172.734,38.053,157.212
C00654=1051.996,306.119,392.995,172.737,38.057,157.213
C00655=1052.002,306.367,392.962,172.740,38.061,157.214
C00656=1052.009,306.615,392.929,172.744,38.064,157.214
C00657=1052.016,306.862,392.897,172.748,38.068,157.215
C00658=1052.023,307.110,392.864,172.752,38.071,157.216
C00659=1052.030,307.357,392.830,172.754,38.075,157.217
C00660=1052.036,307.605,392.798,172.758,38.079,157.218
C00661=1052.043,307.853,392.764,172.762,38.082,157.219
C00662=1052.050,308.100,392.731,172.765,38.085,157.220
C00663=1052.056,308.349,392.698,172.769,38.089,157.221
C00664=1052.063,308.596,392.665,172.772,38.093,157.221
C00665=1052.069,308.843,392.632,172.775,38.096,157.222
C00666=1052.077,309.091,392.599,172.779,38.100,157.223
C00667=1052.083,309.339,392.566,172.783,38.104,157.224
C00668=1052.090,309.586,392.533,172.787,38.107,157.225
C00669=1052.097,309.834,392.500,172.790,38.111,157.226
C00670=1052.104,310.082,392.467,172.793,38.114,157.227
C00671=1052.110,310.329,392.433,172.797,38.118,157.228
C00672=1052.117,310.578,392.400,172.800,38.122,157.228
C00673=1052.124,310.825,392.367,172.804,38.125,157.229
C00674=1052.131,311.073,392.334,172.808,38.129,157.230
C00675=1052.137,311.320,392.300,172.812,38.132,157.231
C00676=1052.144,311.568,392.267,172.815,38.136,157.232
C00677=1052.151,311.816,392.233,172.819,38.140,157.233
C00678=1052.158,312.063,392.200,172.822,38.143,157.234
C00679=1052.165,312.311,392.167,172.825,38.147,157.234
C00680=1052.171,312.559,392.134,172.829,38.150,157.235
C00681=1052.179,312.806,392.101,172.833,38.154,157.236
C00682=1052.186,313.054,392.067,172.837,38.158,157.237
C00683=1052.192,313.302,392.034,172.840,38.162,157.238
C00684=1052.199,313.549,392.000,172.844,38.165,157.239
C00685=1052.205,313.797,391.966,172.848,38.169,157.240
C00686=1052.212,314.044,391.932,172.851,38.173,157.241
C00687=1052.218,314.292,391.898,172.854,38.177,157.242
C00688=1052.225,314.540,391.865,172.858,38.180,157.243
C00689=1052.231,314.787,391.831,172.862,38.184,157.243
C00690=1052.238,315.035,391.797,172.866,38.188,157.244
C00691=1052.244,315.282,391.763,172.869,38.192,157.245
C00692=1052.251,315.530,391.729,172.873,38.196,157.246
C00693=1052.257,315.777,391.695,172.877,38.199,157.247
C00694=1052.264,316.025,391.662,172.880,38.203,157.248
C00695=1052.270,316.273,391.627,172.883,38.207,157.249
C00696=1052.277,316.520,391.594,172.887,38.211,157.250
C00697=1052.283,316.768,391.559,172.891,38.214,157.251
C00698=1052.290,317.015,391.526,172.895,38.218,157.252
C00699=1052.296,317.263,391.492,172.898,38.222,157.253
C00700=1052.304,317.511,391.458,172.902,38.226,157.254
C00701=1052.309,317.758,391.424,172.906,38.230,157.255
C00702=1052.317,318.006,391.390,172.910,38.233,157.255
C00703=1052.324,318.290,391.351,172.914,38.238,157.257
C00704=1052.331,318.574,391.312,172.919,38.242,157.258
C00705=1052.339,318.858,391.273,172.922,38.247,157.259
C00706=1052.347,319.143,391.233,172.926,38.251,157.260
C00707=1052.353,319.390,391.200,172.930,38.255,157.261
C00708=1052.360,319.637,391.164,172.934,38.259,157.262
C00709=1052.367,319.885,391.131,172.938,38.263,157.263
C00710=1052.373,320.132,391.097,172.941,38.267,157.264
C00711=1052.380,320.380,391.063,172.945,38.270,157.265
C00712=1052.387,320.628,391.028,172.949,38.274,157.265
C00713=1052.394,320.876,390.994,172.953,38.278,157.266
C00714=1052.401,321.123,390.959,172.957,38.282,157.267
C00715=1052.407,321.370,390.925,172.960,38.286,157.268
C00716=1052.414,321.618,390.891,172.964,38.290,157.269
C00717=1052.421,321.865,390.856,172.968,38.294,157.270
C00718=1052.428,322.113,390.822,172.972,38.298,157.271
C00719=1052.434,322.361,390.788,172.976,38.302,157.272
C00720=1052.441,322.608,390.755,172.979,38.306,157.273
C00721=1052.448,322.855,390.719,172.983,38.310,157.274
C00722=1052.454,323.103,390.685,172.987,38.314,157.275
C00723=1052.462,323.350,390.650,172.991,38.317,157.276
C00724=1052.468,323.598,390.616,172.995,38.321,157.277
C00725=1052.475,323.846,390.582,172.998,38.325,157.278
C00726=1052.482,324.093,390.547,173.002,38.329,157.279
C00727=1052.489,324.341,390.513,173.006,38.333,157.280
C00728=1052.496,324.588,390.478,173.011,38.337,157.281
C00729=1052.503,324.836,390.444,173.015,38.341,157.282
C00730=1052.509,325.083,390.410,173.019,38.345,157.283
C00731=1052.516,325.331,390.375,173.022,38.349,157.284
C00732=1052.523,325.578,390.340,173.026,38.353,157.285
C00733=1052.530,325.826,390.306,173.030,38.357,157.286
C00734=1052.537,326.073,390.271,173.034,38.360,157.287
C00735=1052.543,326.321,390.237,173.038,38.364,157.288
C00736=1052.551,326.568,390.202,173.041,38.368,157.289
C00737=1052.557,326.815,390.167,173.045,38.372,157.290
C00738=1052.565,327.063,390.133,173.049,38.376,157.291
C00739=1052.571,327.310,390.098,173.054,38.380,157.292
C00740=1052.578,327.558,390.063,173.058,38.384,157.292
C00741=1052.586,327.806,390.029,173.062,38.388,157.294
C00742=1052.593,328.054,389.994,173.065,38.392,157.295
C00743=1052.599,328.301,389.958,173.069,38.396,157.296
C00744=1052.607,328.549,389.925,173.073,38.400,157.296
C00745=1052.613,328.796,389.889,173.077,38.404,157.297
C00746=1052.620,329.043,389.854,173.081,38.408,157.298
C00747=1052.628,329.290,389.820,173.086,38.412,157.300
C00748=1052.634,329.538,389.785,173.089,38.416,157.301
C00749=1052.641,329.786,389.750,173.093,38.420,157.301
C00750=1052.648,330.034,389.715,173.097,38.424,157.302
C00751=1052.655,330.281,389.680,173.101,38.428,157.304
C00752=1052.662,330.529,389.644,173.105,38.432,157.305
C00753=1052.669,330.776,389.609,173.110,38.436,157.305
C00754=1052.675,331.023,389.574,173.114,38.440,157.307
C00755=1052.682,331.271,389.539,173.118,38.444,157.308
C00756=1052.689,331.518,389.504,173.121,38.449,157.309
C00757=1052.696,331.765,389.469,173.125,38.453,157.310
C00758=1052.702,332.013,389.434,173.129,38.457,157.311
C00759=1052.710,332.292,389.394,173.134,38.462,157.312
C00760=1052.718,332.571,389.354,173.139,38.466,157.313
C00761=1052.726,332.850,389.314,173.143,38.471,157.314
C00762=1052.733,333.129,389.275,173.148,38.475,157.315
C00763=1052.741,333.376,389.239,173.152,38.480,157.316
C00764=1052.748,333.623,389.203,173.156,38.484,157.317
C00765=1052.755,333.871,389.168,173.160,38.488,157.319
C00766=1052.761,334.118,389.133,173.165,38.492,157.320
C00767=1052.768,334.366,389.098,173.169,38.497,157.321
C00768=1052.775,334.613,389.061,173.173,38.501,157.322
C00769=1052.782,334.861,389.026,173.176,38.505,157.323
C00770=1052.789,335.108,388.991,173.180,38.509,157.324
C00771=1052.795,335.355,388.956,173.185,38.513,157.325
C00772=1052.803,335.603,388.920,173.189,38.518,157.326
C00773=1052.810,335.850,388.884,173.193,38.522,157.327
C00774=1052.817,336.097,388.849,173.197,38.526,157.328
C00775=1052.824,336.345,388.813,173.202,38.530,157.329
C00776=1052.830,336.593,388.777,173.206,38.535,157.330
C00777=1052.837,336.839,388.741,173.210,38.539,157.331
C00778=1052.844,337.087,388.706,173.214,38.543,157.332
C00779=1052.852,337.334,388.670,173.219,38.547,157.333
C00780=1052.858,337.582,388.634,173.223,38.552,157.335
C00781=1052.865,337.829,388.599,173.227,38.556,157.336
C00782=1052.872,338.077,388.563,173.232,38.560,157.337
C00783=1052.879,338.324,388.527,173.235,38.565,157.338
C00784=1052.886,338.570,388.491,173.239,38.569,157.339
C00785=1052.893,338.819,388.455,173.243,38.573,157.340
C00786=1052.899,339.066,388.419,173.248,38.578,157.341
C00787=1052.906,339.313,388.384,173.252,38.582,157.342
C00788=1052.914,339.560,388.347,173.256,38.586,157.343
C00789=1052.920,339.807,388.311,173.261,38.590,157.344
C00790=1052.927,340.054,388.275,173.265,38.595,157.345
C00791=1052.935,340.302,388.240,173.269,38.599,157.347
C00792=1052.941,340.549,388.203,173.274,38.604,157.348
C00793=1052.949,340.797,388.167,173.278,38.608,157.349
C00794=1052.955,341.044,388.131,173.282,38.613,157.350
C00795=1052.962,341.292,388.095,173.287,38.617,157.351
C00796=1052.969,341.539,388.059,173.291,38.621,157.352
C00797=1052.976,341.786,388.022,173.295,38.626,157.353
C00798=1052.983,342.033,387.987,173.300,38.630,157.354
C00799=1052.991,342.281,387.950,173.304,38.635,157.356
C00800=1052.997,342.528,387.914,173.308,38.639,157.357
C00801=1053.005,342.776,387.878,173.313,38.643,157.358
C00802=1053.011,343.023,387.842,173.317,38.648,157.359
C00803=1053.019,343.270,387.806,173.322,38.652,157.360
C00804=1053.025,343.517,387.769,173.326,38.657,157.361
C00805=1053.033,343.764,387.732,173.330,38.661,157.362
C00806=1053.039,344.011,387.696,173.335,38.666,157.364
C00807=1053.046,344.259,387.659,173.339,38.670,157.365
C00808=1053.053,344.506,387.623,173.344,38.675,157.366
C00809=1053.060,344.753,387.586,173.348,38.679,157.367
C00810=1053.067,345.000,387.551,173.352,38.684,157.368
C00811=1053.074,345.248,387.514,173.357,38.688,157.369
C00812=1053.081,345.495,387.477,173.361,38.693,157.370
C00813=1053.089,345.742,387.440,173.366,38.697,157.372
C00814=1053.096,345.990,387.404,173.370,38.702,157.373
C00815=1053.104,346.264,387.363,173.375,38.707,157.374
C00816=1053.111,346.539,387.323,173.380,38.712,157.375
C00817=1053.119,346.815,387.281,173.385,38.718,157.377
C00818=1053.127,347.089,387.241,173.390,38.723,157.378
C00819=1053.133,347.336,387.204,173.395,38.727,157.379
C00820=1053.141,347.583,387.167,173.399,38.732,157.380
C00821=1053.148,347.831,387.131,173.404,38.736,157.382
C00822=1053.155,348.077,387.093,173.408,38.741,157.383
C00823=1053.162,348.325,387.057,173.413,38.746,157.384
C00824=1053.169,348.572,387.020,173.417,38.750,157.385
C00825=1053.177,348.820,386.983,173.422,38.755,157.386
C00826=1053.183,349.067,386.946,173.426,38.759,157.387
C00827=1053.190,349.314,386.909,173.431,38.764,157.389
C00828=1053.198,349.561,386.873,173.435,38.769,157.390
C00829=1053.204,349.808,386.836,173.440,38.773,157.391
C00830=1053.212,350.055,386.798,173.445,38.778,157.392
C00831=1053.219,350.303,386.761,173.450,38.783,157.394
C00832=1053.227,350.549,386.724,173.454,38.788,157.395
C00833=1053.234,350.797,386.687,173.459,38.792,157.396
C00834=1053.240,351.044,386.650,173.463,38.797,157.397
C00835=1053.247,351.291,386.613,173.468,38.802,157.398
C00836=1053.254,351.538,386.576,173.472,38.806,157.400
C00837=1053.262,351.786,386.538,173.477,38.811,157.401
C00838=1053.269,352.033,386.501,173.481,38.816,157.402
C00839=1053.276,352.279,386.464,173.486,38.821,157.403
C00840=1053.284,352.526,386.427,173.492,38.826,157.405
C00841=1053.290,352.774,386.390,173.496,38.830,157.406
C00842=1053.298,353.021,386.352,173.501,38.835,157.407
C00843=1053.305,353.268,386.315,173.505,38.840,157.408
C00844=1053.312,353.515,386.277,173.510,38.845,157.410
C00845=1053.319,353.762,386.240,173.514,38.850,157.411
C00846=1053.326,354.009,386.203,173.519,38.855,157.412
C00847=1053.333,354.256,386.165,173.524,38.860,157.413
C00848=1053.341,354.503,386.128,173.528,38.864,157.415
C00849=1053.348,354.750,386.090,173.534,38.869,157.416
C00850=1053.355,354.997,386.053,173.538,38.874,157.417
C00851=1053.362,355.244,386.015,173.543,38.879,157.418
C00852=1053.370,355.492,385.978,173.548,38.884,157.420
C00853=1053.377,355.739,385.940,173.552,38.889,157.421
C00854=1053.384,355.986,385.903,173.557,38.894,157.422
C00855=1053.391,356.233,385.864,173.563,38.898,157.424
C00856=1053.398,356.480,385.827,173.567,38.903,157.425
C00857=1053.405,356.727,385.789,173.572,38.909,157.426
C00858=1053.413,356.974,385.751,173.577,38.914,157.428
C00859=1053.420,357.221,385.714,173.581,38.919,157.429
C00860=1053.427,357.468,385.676,173.587,38.924,157.430
C00861=1053.434,357.715,385.639,173.592,38.928,157.431
C00862=1053.442,357.962,385.600,173.596,38.933,157.433
C00863=1053.449,358.209,385.563,173.601,38.938,157.434
C00864=1053.457,358.456,385.525,173.606,38.944,157.435
C00865=1053.463,358.703,385.486,173.610,38.949,157.437
C00866=1053.470,358.950,385.449,173.616,38.953,157.438
C00867=1053.478,359.197,385.411,173.621,38.959,157.439
C00868=1053.485,359.444,385.373,173.625,38.964,157.441
C00869=1053.492,359.691,385.334,173.630,38.969,157.442
C00870=1053.499,359.938,385.297,173.636,38.974,157.443
C00871=1053.508,360.218,385.253,173.641,38.979,157.445
C00872=1053.516,360.498,385.210,173.646,38.985,157.446
C00873=1053.525,360.778,385.166,173.653,38.991,157.448
C00874=1053.533,361.058,385.124,173.658,38.997,157.449
C00875=1053.540,361.305,385.085,173.663,39.002,157.451
C00876=1053.548,361.551,385.047,173.668,39.007,157.452
C00877=1053.555,361.798,385.010,173.673,39.013,157.453
C00878=1053.562,362.045,384.971,173.678,39.017,157.455
C00879=1053.570,362.292,384.932,173.683,39.023,157.456
C00880=1053.577,362.540,384.895,173.688,39.028,157.458
C00881=1053.584,362.786,384.856,173.693,39.033,157.459
C00882=1053.592,363.033,384.818,173.698,39.039,157.460
C00883=1053.600,363.280,384.779,173.703,39.043,157.462
C00884=1053.607,363.527,384.740,173.709,39.049,157.463
C00885=1053.614,363.773,384.702,173.713,39.054,157.465
C00886=1053.621,364.021,384.664,173.718,39.060,157.466
C00887=1053.629,364.268,384.625,173.724,39.065,157.467
C00888=1053.636,364.515,384.586,173.729,39.070,157.469
C00889=1053.642,364.762,384.548,173.734,39.075,157.470
C00890=1053.650,365.008,384.509,173.739,39.081,157.472
C00891=1053.657,365.256,384.470,173.744,39.086,157.473
C00892=1053.665,365.502,384.431,173.749,39.092,157.474
C00893=1053.672,365.749,384.392,173.755,39.097,157.476
C00894=1053.680,365.996,384.354,173.760,39.102,157.477
C00895=1053.687,366.243,384.315,173.765,39.108,157.479
C00896=1053.695,366.489,384.277,173.770,39.113,157.480
C00897=1053.702,366.737,384.237,173.775,39.119,157.482
C00898=1053.709,366.983,384.199,173.780,39.124,157.483
C00899=1053.717,367.229,384.160,173.786,39.129,157.484
C00900=1053.724,367.477,384.120,173.791,39.135,157.486
C00901=1053.732,367.723,384.082,173.796,39.140,157.487
C00902=1053.739,367.971,384.043,173.802,39.146,157.489
C00903=1053.746,368.217,384.003,173.807,39.151,157.490
C00904=1053.754,368.464,383.965,173.812,39.156,157.492
C00905=1053.761,368.711,383.925,173.818,39.162,157.493
C00906=1053.769,368.957,383.887,173.822,39.168,157.495
C00907=1053.776,369.205,383.848,173.828,39.173,157.496
C00908=1053.783,369.451,383.808,173.833,39.178,157.498
C00909=1053.792,369.698,383.770,173.838,39.184,157.499
C00910=1053.799,369.944,383.730,173.844,39.190,157.501
C00911=1053.806,370.192,383.691,173.849,39.195,157.502
C00912=1053.814,370.438,383.652,173.854,39.200,157.504
C00913=1053.821,370.685,383.613,173.860,39.206,157.505
C00914=1053.830,370.932,383.573,173.865,39.212,157.507
C00915=1053.837,371.179,383.535,173.871,39.218,157.508
C00916=1053.844,371.425,383.495,173.876,39.223,157.510
C00917=1053.853,371.672,383.455,173.881,39.228,157.511
C00918=1053.860,371.919,383.416,173.887,39.234,157.513
C00919=1053.867,372.166,383.377,173.892,39.240,157.514
C00920=1053.875,372.412,383.337,173.898,39.246,157.516
C00921=1053.882,372.659,383.297,173.903,39.251,157.517
C00922=1053.889,372.905,383.258,173.909,39.257,157.519
C00923=1053.897,373.152,383.218,173.914,39.263,157.520
C00924=1053.904,373.400,383.178,173.920,39.269,157.522
C00925=1053.912,373.646,383.139,173.925,39.275,157.523
C00926=1053.919,373.893,383.099,173.931,39.280,157.525
C00927=1053.929,374.191,383.051,173.937,39.287,157.527
C00928=1053.938,374.490,383.002,173.944,39.294,157.529
C00929=1053.947,374.788,382.955,173.951,39.301,157.531
C00930=1053.956,375.087,382.906,173.958,39.308,157.533
C00931=1053.964,375.334,382.866,173.963,39.314,157.534
C00932=1053.971,375.581,382.826,173.969,39.320,157.536
C00933=1053.979,375.827,382.787,173.975,39.326,157.537
C00934=1053.987,376.074,382.747,173.980,39.332,157.539
C00935=1053.995,376.321,382.707,173.986,39.338,157.541
C00936=1054.002,376.568,382.667,173.992,39.344,157.542
C00937=1054.010,376.814,382.626,173.998,39.349,157.544
C00938=1054.018,377.060,382.587,174.003,39.355,157.545
C00939=1054.025,377.307,382.547,174.009,39.361,157.547
C00940=1054.033,377.553,382.506,174.014,39.367,157.549
C00941=1054.041,377.800,382.466,174.020,39.373,157.550
C00942=1054.049,378.047,382.427,174.025,39.379,157.552
C00943=1054.057,378.293,382.386,174.032,39.385,157.554
C00944=1054.065,378.540,382.346,174.038,39.391,157.555
C00945=1054.072,378.786,382.306,174.043,39.397,157.557
C00946=1054.080,379.033,382.266,174.049,39.403,157.558
C00947=1054.087,379.280,382.226,174.054,39.409,157.560
C00948=1054.095,379.526,382.185,174.061,39.415,157.562
C00949=1054.102,379.773,382.145,174.066,39.421,157.563
C00950=1054.110,380.019,382.104,174.072,39.427,157.565
C00951=1054.118,380.266,382.063,174.078,39.433,157.567
C00952=1054.126,380.513,382.024,174.084,39.440,157.568
C00953=1054.134,380.759,381.983,174.090,39.446,157.570
C00954=1054.141,381.006,381.942,174.096,39.452,157.572
C00955=1054.150,381.252,381.901,174.101,39.458,157.573
C00956=1054.157,381.499,381.861,174.107,39.464,157.575
C00957=1054.165,381.745,381.820,174.114,39.471,157.577
C00958=1054.173,381.992,381.779,174.119,39.477,157.579
C00959=1054.181,382.238,381.739,174.125,39.483,157.580
C00960=1054.188,382.484,381.697,174.132,39.489,157.582
C00961=1054.196,382.731,381.657,174.137,39.496,157.584
C00962=1054.204,382.977,381.616,174.143,39.502,157.586
C00963=1054.211,383.224,381.575,174.149,39.508,157.587
C00964=1054.219,383.470,381.534,174.155,39.514,157.589
C00965=1054.227,383.716,381.493,174.161,39.521,157.591
C00966=1054.235,383.963,381.452,174.167,39.527,157.593
C00967=1054.243,384.210,381.411,174.173,39.533,157.594
C00968=1054.250,384.456,381.370,174.179,39.540,157.596
C00969=1054.258,384.703,381.330,174.185,39.546,157.598
C00970=1054.266,384.949,381.289,174.192,39.552,157.600
C00971=1054.274,385.195,381.247,174.197,39.559,157.601
C00972=1054.282,385.441,381.206,174.203,39.566,157.603
C00973=1054.290,385.688,381.165,174.210,39.572,157.605
C00974=1054.298,385.935,381.124,174.216,39.578,157.607
C00975=1054.306,386.180,381.083,174.222,39.585,157.609
C00976=1054.314,386.427,381.042,174.228,39.591,157.610
C00977=1054.322,386.674,381.001,174.235,39.598,157.612
C00978=1054.330,386.920,380.959,174.241,39.604,157.614
C00979=1054.338,387.166,380.918,174.246,39.611,157.616
C00980=1054.346,387.412,380.877,174.253,39.618,157.618
C00981=1054.354,387.659,380.835,174.259,39.624,157.619
C00982=1054.362,387.905,380.794,174.266,39.630,157.621
C00983=1054.373,388.236,380.738,174.274,39.639,157.624
C00984=1054.384,388.567,380.682,174.283,39.648,157.626
C00985=1054.394,388.898,380.627,174.291,39.657,157.629
C00986=1054.406,389.229,380.571,174.300,39.666,157.631
C00987=1054.414,389.475,380.529,174.306,39.673,157.633
C00988=1054.422,389.722,380.488,174.312,39.679,157.635
C00989=1054.430,389.968,380.446,174.318,39.686,157.637
C00990=1054.438,390.214,380.404,174.325,39.693,157.639
C00991=1054.447,390.460,380.363,174.331,39.699,157.641
C00992=1054.454,390.706,380.321,174.338,39.706,157.643
C00993=1054.462,390.953,380.278,174.345,39.713,157.644
C00994=1054.471,391.198,380.237,174.351,39.720,157.646
C00995=1054.479,391.445,380.195,174.358,39.727,157.648
C00996=1054.486,391.691,380.153,174.364,39.734,157.650
C00997=1054.495,391.937,380.111,174.371,39.740,157.652
C00998=1054.503,392.183,380.069,174.376,39.747,157.654
C00999=1054.511,392.430,380.027,174.383,39.754,157.656
C01000=1054.519,392.676,379.985,174.390,39.761,157.658
C01001=1054.528,392.922,379.943,174.396,39.768,157.660
C01002=1054.536,393.169,379.901,174.403,39.775,157.662
C01003=1054.543,393.415,379.859,174.409,39.782,157.664
C01004=1054.552,393.661,379.816,174.416,39.789,157.666
C01005=1054.560,393.907,379.774,174.423,39.796,157.668
C01006=1054.568,394.154,379.732,174.429,39.803,157.670
C01007=1054.576,394.400,379.689,174.436,39.810,157.672
C01008=1054.585,394.645,379.647,174.443,39.817,157.674
C01009=1054.593,394.892,379.605,174.449,39.824,157.676
C01010=1054.601,395.138,379.562,174.456,39.831,157.678
C01011=1054.609,395.384,379.520,174.463,39.838,157.680
C01012=1054.617,395.630,379.477,174.470,39.846,157.682
C01013=1054.626,395.877,379.435,174.476,39.852,157.684
C01014=1054.634,396.123,379.392,174.484,39.860,157.686
C01015=1054.642,396.369,379.350,174.491,39.867,157.688
C01016=1054.650,396.615,379.307,174.497,39.874,157.690
C01017=1054.658,396.861,379.264,174.504,39.881,157.692
C01018=1054.667,397.108,379.221,174.511,39.889,157.694
C01019=1054.675,397.354,379.178,174.518,39.896,157.696
C01020=1054.684,397.600,379.135,174.525,39.903,157.698
C01021=1054.692,397.846,379.093,174.531,39.911,157.700
C01022=1054.700,398.092,379.050,174.538,39.918,157.703
C01023=1054.709,398.338,379.007,174.545,39.925,157.705
C01024=1054.717,398.584,378.964,174.553,39.932,157.707
C01025=1054.726,398.830,378.921,174.559,39.940,157.709
C01026=1054.734,399.076,378.878,174.566,39.948,157.711
C01027=1054.743,399.322,378.835,174.573,39.955,157.713
C01028=1054.750,399.568,378.791,174.580,39.962,157.715
C01029=1054.759,399.814,378.748,174.587,39.970,157.717
C01030=1054.767,400.060,378.705,174.595,39.977,157.720
C01031=1054.776,400.306,378.662,174.602,39.985,157.722
C01032=1054.784,400.553,378.619,174.608,39.992,157.724
C01033=1054.793,400.799,378.576,174.615,40.000,157.726
C01034=1054.801,401.045,378.533,174.623,40.007,157.728
C01035=1054.809,401.290,378.489,174.630,40.015,157.731
C01036=1054.818,401.536,378.446,174.637,40.022,157.733
C01037=1054.827,401.783,378.403,174.644,40.030,157.735
C01038=1054.835,402.029,378.359,174.652,40.038,157.737
C01039=1054.849,402.428,378.288,174.663,40.050,157.741
C01040=1054.863,402.827,378.218,174.675,40.062,157.744
C01041=1054.877,403.227,378.147,174.687,40.075,157.748
C01042=1054.890,403.626,378.076,174.699,40.088,157.752
C01043=1054.899,403.873,378.032,174.706,40.096,157.754
C01044=1054.908,404.118,377.988,174.713,40.103,157.756
C01045=1054.916,404.363,377.945,174.721,40.111,157.758
C01046=1054.924,404.610,377.901,174.728,40.119,157.761
C01047=1054.934,404.856,377.857,174.735,40.127,157.763
C01048=1054.942,405.102,377.813,174.744,40.135,157.765
C01049=1054.951,405.348,377.769,174.751,40.143,157.768
C01050=1054.959,405.594,377.725,174.759,40.151,157.770
C01051=1054.968,405.840,377.681,174.766,40.159,157.772
C01052=1054.976,406.086,377.636,174.774,40.167,157.775
C01053=1054.985,406.332,377.593,174.781,40.175,157.777
C01054=1054.993,406.577,377.548,174.788,40.183,157.779
C01055=1055.002,406.824,377.504,174.796,40.191,157.782
C01056=1055.011,407.069,377.460,174.803,40.199,157.784
C01057=1055.019,407.316,377.415,174.812,40.207,157.786
C01058=1055.028,407.561,377.371,174.819,40.215,157.789
C01059=1055.037,407.807,377.327,174.827,40.224,157.791
C01060=1055.045,408.053,377.282,174.835,40.232,157.794
C01061=1055.055,408.299,377.238,174.842,40.240,157.796
C01062=1055.063,408.544,377.193,174.850,40.248,157.799
C01063=1055.071,408.791,377.148,174.858,40.256,157.801
C01064=1055.080,409.036,377.104,174.866,40.264,157.803
C01065=1055.089,409.282,377.059,174.873,40.273,157.806
C01066=1055.098,409.528,377.015,174.882,40.281,157.808
C01067=1055.107,409.773,376.970,174.889,40.290,157.811
C01068=1055.116,410.020,376.925,174.897,40.298,157.813
C01069=1055.125,410.265,376.881,174.905,40.306,157.816
C01070=1055.133,410.511,376.836,174.913,40.314,157.818
C01071=1055.142,410.757,376.791,174.921,40.323,157.821
C01072=1055.152,411.003,376.747,174.930,40.331,157.823
C01073=1055.161,411.249,376.701,174.937,40.340,157.826
C01074=1055.169,411.495,376.657,174.945,40.348,157.828
C01075=1055.178,411.740,376.612,174.953,40.356,157.831
C01076=1055.187,411.986,376.567,174.961,40.365,157.833
C01077=1055.196,412.232,376.521,174.969,40.373,157.836
C01078=1055.205,412.478,376.477,174.978,40.382,157.838
C01079=1055.215,412.724,376.432,174.985,40.391,157.841
C01080=1055.224,412.970,376.386,174.994,40.400,157.844
C01081=1055.232,413.215,376.341,175.002,40.408,157.846
C01082=1055.242,413.460,376.297,175.011,40.416,157.849
C01083=1055.251,413.706,376.251,175.018,40.425,157.851
C01084=1055.260,413.952,376.206,175.027,40.434,157.854
C01085=1055.269,414.198,376.160,175.035,40.443,157.857
C01086=1055.278,414.444,376.115,175.044,40.452,157.859
C01087=1055.287,414.689,376.069,175.052,40.461,157.862
C01088=1055.296,414.935,376.023,175.061,40.469,157.865
C01089=1055.305,415.180,375.978,175.068,40.479,157.867
C01090=1055.314,415.426,375.932,175.077,40.487,157.870
C01091=1055.328,415.816,375.859,175.091,40.502,157.874
C01092=1055.342,416.207,375.787,175.104,40.515,157.878
C01093=1055.356,416.562,375.721,175.117,40.529,157.882
C01094=1055.369,416.916,375.655,175.129,40.541,157.886
C01095=1055.383,417.270,375.589,175.141,40.555,157.890
C01096=1055.396,417.625,375.522,175.155,40.568,157.894
C01097=1055.405,417.871,375.476,175.163,40.577,157.897
C01098=1055.415,418.116,375.430,175.172,40.586,157.900
C01099=1055.424,418.362,375.384,175.181,40.595,157.903
C01100=1055.433,418.608,375.338,175.190,40.604,157.905
C01101=1055.443,418.853,375.292,175.198,40.614,157.908
C01102=1055.452,419.098,375.245,175.207,40.623,157.911
C01103=1055.462,419.344,375.199,175.216,40.632,157.914
C01104=1055.470,419.589,375.152,175.225,40.642,157.917
C01105=1055.480,419.835,375.106,175.234,40.651,157.920
C01106=1055.490,420.080,375.060,175.243,40.660,157.923
C01107=1055.499,420.326,375.013,175.251,40.670,157.925
C01108=1055.507,420.571,374.967,175.261,40.679,157.928
C01109=1055.517,420.817,374.920,175.270,40.688,157.931
C01110=1055.527,421.062,374.874,175.279,40.698,157.934
C01111=1055.536,421.308,374.826,175.288,40.707,157.937
C01112=1055.545,421.553,374.780,175.297,40.717,157.940
C01113=1055.555,421.799,374.734,175.307,40.727,157.943
C01114=1055.564,422.044,374.686,175.316,40.736,157.946
C01115=1055.574,422.290,374.640,175.325,40.746,157.949
C01116=1055.584,422.534,374.593,175.334,40.756,157.952
C01117=1055.593,422.781,374.546,175.344,40.765,157.955
C01118=1055.602,423.025,374.499,175.353,40.775,157.958
C01119=1055.611,423.271,374.452,175.362,40.785,157.961
C01120=1055.622,423.517,374.405,175.372,40.794,157.964
C01121=1055.631,423.761,374.358,175.381,40.804,157.967
C01122=1055.640,424.007,374.311,175.390,40.814,157.970
C01123=1055.651,424.253,374.263,175.401,40.824,157.973
C01124=1055.659,424.498,374.216,175.410,40.834,157.976
C01125=1055.670,424.743,374.169,175.419,40.843,157.979
C01126=1055.680,424.988,374.121,175.429,40.853,157.982
C01127=1055.689,425.234,374.074,175.438,40.863,157.985
C01128=1055.699,425.478,374.027,175.448,40.874,157.989
C01129=1055.708,425.724,373.979,175.458,40.884,157.992
C01130=1055.719,425.969,373.932,175.468,40.894,157.995
C01131=1055.728,426.215,373.884,175.477,40.904,157.998
C01132=1055.738,426.460,373.837,175.487,40.914,158.001
C01133=1055.748,426.706,373.789,175.497,40.924,158.004
C01134=1055.757,426.951,373.740,175.507,40.934,158.007
C01135=1055.767,427.195,373.694,175.517,40.944,158.011
C01136=1055.776,427.441,373.646,175.527,40.954,158.014
C01137=1055.787,427.686,373.598,175.537,40.965,158.017
C01138=1055.796,427.931,373.550,175.546,40.975,158.020
C01139=1055.806,428.176,373.502,175.557,40.985,158.024
C01140=1055.816,428.421,373.454,175.567,40.996,158.027
C01141=1055.826,428.666,373.406,175.577,41.006,158.030
C01142=1055.836,428.912,373.358,175.587,41.016,158.033
C01143=1055.846,429.157,373.310,175.598,41.027,158.037
C01144=1055.856,429.402,373.261,175.607,41.037,158.040
C01145=1055.866,429.647,373.213,175.618,41.048,158.043
C01146=1055.876,429.893,373.165,175.628,41.058,158.047
C01147=1055.886,430.138,373.117,175.639,41.069,158.050
C01148=1055.896,430.383,373.068,175.649,41.080,158.054
C01149=1055.911,430.759,372.993,175.665,41.096,158.059
C01150=1055.926,431.135,372.919,175.681,41.113,158.064
C01151=1055.942,431.512,372.844,175.697,41.129,158.069
C01152=1055.957,431.888,372.769,175.713,41.145,158.075
C01153=1055.967,432.134,372.720,175.724,41.156,158.078
C01154=1055.978,432.378,372.671,175.734,41.167,158.082
C01155=1055.987,432.623,372.623,175.745,41.178,158.085
C01156=1055.998,432.869,372.574,175.756,41.189,158.089
C01157=1056.008,433.113,372.525,175.767,41.200,158.092
C01158=1056.017,433.358,372.476,175.778,41.211,158.096
C01159=1056.028,433.603,372.426,175.789,41.222,158.099
C01160=1056.039,433.847,372.378,175.800,41.233,158.103
C01161=1056.049,434.093,372.329,175.811,41.245,158.107
C01162=1056.059,434.337,372.280,175.822,41.255,158.110
C01163=1056.070,434.582,372.230,175.833,41.267,158.114
C01164=1056.080,434.828,372.181,175.844,41.278,158.117
C01165=1056.090,435.072,372.132,175.854,41.289,158.121
C01166=1056.101,435.317,372.082,175.866,41.300,158.125
C01167=1056.111,435.562,372.033,175.877,41.312,158.128
C01168=1056.122,435.807,371.983,175.888,41.323,158.132
C01169=1056.133,436.052,371.934,175.899,41.334,158.136
C01170=1056.143,436.296,371.885,175.911,41.346,158.139
C01171=1056.153,436.541,371.835,175.923,41.357,158.143
C01172=1056.164,436.786,371.785,175.934,41.369,158.147
C01173=1056.175,437.031,371.735,175.946,41.380,158.151
C01174=1056.186,437.276,371.685,175.957,41.392,158.155
C01175=1056.195,437.520,371.635,175.968,41.403,158.158
C01176=1056.206,437.765,371.585,175.980,41.415,158.162
C01177=1056.217,438.010,371.536,175.991,41.427,158.166
C01178=1056.228,438.254,371.485,176.004,41.439,158.170
C01179=1056.238,438.499,371.435,176.015,41.450,158.174
C01180=1056.248,438.744,371.385,176.027,41.462,158.178
C01181=1056.259,438.989,371.334,176.038,41.474,158.182
C01182=1056.270,439.233,371.284,176.051,41.486,158.186
C01183=1056.281,439.478,371.235,176.062,41.497,158.189
C01184=1056.291,439.723,371.184,176.074,41.510,158.193
C01185=1056.302,439.967,371.133,176.087,41.521,158.197
C01186=1056.313,440.212,371.083,176.098,41.533,158.201
C01187=1056.323,440.456,371.032,176.111,41.545,158.205
C01188=1056.334,440.701,370.982,176.123,41.557,158.209
C01189=1056.345,440.945,370.931,176.135,41.570,158.213
C01190=1056.356,441.189,370.880,176.147,41.582,158.218
C01191=1056.367,441.434,370.829,176.159,41.594,158.222
C01192=1056.378,441.679,370.778,176.172,41.606,158.226
C01193=1056.389,441.924,370.728,176.185,41.618,158.230
C01194=1056.400,442.168,370.677,176.197,41.631,158.234
C01195=1056.410,442.412,370.626,176.210,41.643,158.238
C01196=1056.422,442.657,370.574,176.222,41.656,158.242
C01197=1056.432,442.902,370.524,176.234,41.668,158.246
C01198=1056.444,443.145,370.473,176.247,41.680,158.251
C01199=1056.455,443.390,370.421,176.259,41.693,158.255
C01200=1056.466,443.635,370.370,176.272,41.706,158.259
C01201=1056.477,443.879,370.318,176.285,41.718,158.263
C01202=1056.488,444.123,370.267,176.299,41.731,158.268
C01203=1056.499,444.368,370.215,176.312,41.743,158.272
C01204=1056.511,444.612,370.164,176.324,41.756,158.276
C01205=1056.529,445.010,370.080,176.345,41.777,158.283
C01206=1056.547,445.406,369.996,176.366,41.797,158.290
C01207=1056.565,445.804,369.912,176.388,41.818,158.298
C01208=1056.584,446.202,369.827,176.410,41.840,158.305
C01209=1056.596,446.445,369.776,176.423,41.853,158.309
C01210=1056.607,446.688,369.724,176.436,41.866,158.314
C01211=1056.619,446.932,369.673,176.450,41.879,158.318
C01212=1056.631,447.176,369.622,176.464,41.891,158.323
C01213=1056.645,447.419,369.571,176.477,41.904,158.327
C01214=1056.659,447.663,369.521,176.491,41.915,158.331
C01215=1056.674,447.907,369.471,176.504,41.928,158.336
C01216=1056.690,448.152,369.423,176.519,41.940,158.340
C01217=1056.707,448.396,369.375,176.533,41.952,158.344
C01218=1056.724,448.641,369.328,176.546,41.963,158.348
C01219=1056.742,448.885,369.280,176.560,41.975,158.352
C01220=1056.762,449.130,369.235,176.575,41.986,158.356
C01221=1056.781,449.375,369.189,176.589,41.997,158.360
C01222=1056.802,449.621,369.143,176.603,42.007,158.364
C01223=1056.824,449.866,369.099,176.617,42.018,158.368
C01224=1056.846,450.111,369.055,176.632,42.028,158.372
C01225=1056.521,450.128,368.769,176.629,42.133,158.401
C01226=1056.499,449.883,368.812,176.614,42.123,158.398
C01227=1056.477,449.637,368.857,176.600,42.113,158.394
C01228=1056.457,449.393,368.902,176.586,42.102,158.390
C01229=1056.435,449.147,368.948,176.571,42.091,158.386
C01230=1056.417,448.902,368.994,176.557,42.080,158.382
C01231=1056.398,448.658,369.041,176.543,42.069,158.378
C01232=1056.381,448.413,369.089,176.528,42.057,158.373
C01233=1056.363,448.168,369.137,176.514,42.046,158.369
C01234=1056.348,447.924,369.185,176.501,42.034,158.365
C01235=1056.332,447.680,369.234,176.487,42.022,158.361
C01236=1056.317,447.436,369.284,176.473,42.010,158.357
C01237=1056.305,447.193,369.334,176.460,41.998,158.352
C01238=1056.291,446.948,369.385,176.445,41.985,158.348
C01239=1056.279,446.705,369.436,176.432,41.972,158.343
C01240=1056.268,446.461,369.489,176.419,41.959,158.339
C01241=1056.257,446.218,369.540,176.405,41.946,158.334
C01242=1056.239,445.841,369.621,176.385,41.926,158.327
C01243=1056.221,445.462,369.701,176.364,41.907,158.321
C01244=1056.203,445.083,369.781,176.344,41.886,158.314
C01245=1056.186,444.705,369.860,176.324,41.867,158.307
C01246=1056.175,444.461,369.912,176.310,41.854,158.303
C01247=1056.164,444.216,369.963,176.297,41.841,158.298
C01248=1056.153,443.972,370.015,176.284,41.829,158.294
C01249=1056.141,443.728,370.067,176.271,41.816,158.290
C01250=1056.131,443.483,370.118,176.258,41.804,158.286
C01251=1056.119,443.239,370.170,176.246,41.791,158.281
C01252=1056.108,442.995,370.221,176.233,41.779,158.277
C01253=1056.097,442.750,370.272,176.220,41.767,158.273
C01254=1056.086,442.506,370.324,176.208,41.754,158.269
C01255=1056.075,442.261,370.374,176.195,41.742,158.264
C01256=1056.064,442.016,370.426,176.182,41.730,158.260
C01257=1056.053,441.772,370.476,176.170,41.718,158.256
C01258=1056.042,441.528,370.527,176.157,41.706,158.252
C01259=1056.031,441.283,370.578,176.145,41.693,158.248
C01260=1056.020,441.038,370.629,176.133,41.681,158.244
C01261=1056.010,440.793,370.680,176.120,41.669,158.240
C01262=1055.999,440.549,370.730,176.108,41.657,158.236
C01263=1055.987,440.305,370.781,176.096,41.645,158.232
C01264=1055.977,440.060,370.832,176.084,41.633,158.228
C01265=1055.966,439.816,370.882,176.072,41.621,158.224
C01266=1055.955,439.572,370.933,176.059,41.609,158.220
C01267=1055.945,439.326,370.983,176.048,41.597,158.216
C01268=1055.934,439.082,371.033,176.036,41.586,158.212
C01269=1055.923,438.837,371.083,176.023,41.574,158.208
C01270=1055.912,438.593,371.134,176.012,41.562,158.204
C01271=1055.902,438.348,371.183,176.000,41.550,158.200
C01272=1055.891,438.103,371.234,175.988,41.539,158.196
C01273=1055.880,437.859,371.285,175.976,41.527,158.192
C01274=1055.870,437.614,371.334,175.965,41.515,158.189
C01275=1055.859,437.369,371.384,175.953,41.504,158.185
C01276=1055.849,437.125,371.434,175.942,41.492,158.181
C01277=1055.838,436.880,371.483,175.930,41.481,158.177
C01278=1055.827,436.635,371.533,175.918,41.470,158.174
C01279=1055.816,436.390,371.583,175.907,41.458,158.170
C01280=1055.806,436.145,371.633,175.895,41.447,158.166
C01281=1055.796,435.901,371.682,175.884,41.435,158.162
C01282=1055.785,435.656,371.732,175.873,41.424,158.158
C01283=1055.774,435.411,371.781,175.861,41.413,158.155
C01284=1055.764,435.166,371.831,175.850,41.402,158.151
C01285=1055.754,434.921,371.880,175.839,41.390,158.148
C01286=1055.743,434.676,371.930,175.828,41.379,158.144
C01287=1055.733,434.432,371.979,175.816,41.368,158.140
C01288=1055.723,434.186,372.028,175.805,41.357,158.137
C01289=1055.712,433.942,372.077,175.794,41.346,158.133
C01290=1055.702,433.697,372.127,175.784,41.335,158.129
C01291=1055.692,433.452,372.175,175.773,41.324,158.126
C01292=1055.681,433.207,372.225,175.762,41.313,158.122
C01293=1055.671,432.963,372.274,175.751,41.302,158.119
C01294=1055.661,432.717,372.323,175.740,41.291,158.115
C01295=1055.651,432.472,372.372,175.730,41.280,158.112
C01296=1055.641,432.228,372.421,175.719,41.269,158.108
C01297=1055.631,431.982,372.470,175.707,41.258,158.105
C01298=1055.615,431.604,372.544,175.691,41.242,158.099
C01299=1055.599,431.226,372.620,175.674,41.225,158.094
C01300=1055.584,430.847,372.696,175.658,41.209,158.089
C01301=1055.568,430.468,372.771,175.642,41.192,158.083
C01302=1055.559,430.223,372.820,175.631,41.182,158.080
C01303=1055.549,429.978,372.868,175.622,41.171,158.077
C01304=1055.539,429.733,372.915,175.611,41.161,158.073
C01305=1055.528,429.488,372.964,175.601,41.150,158.070
C01306=1055.519,429.243,373.013,175.590,41.140,158.067
C01307=1055.508,428.998,373.061,175.580,41.130,158.063
C01308=1055.499,428.752,373.109,175.570,41.119,158.060
C01309=1055.489,428.507,373.157,175.560,41.109,158.057
C01310=1055.478,428.263,373.205,175.549,41.098,158.053
C01311=1055.469,428.017,373.253,175.539,41.088,158.050
C01312=1055.459,427.772,373.301,175.529,41.078,158.047
C01313=1055.449,427.527,373.349,175.519,41.068,158.044
C01314=1055.439,427.282,373.397,175.509,41.057,158.040
C01315=1055.429,427.037,373.444,175.499,41.047,158.037
C01316=1055.420,426.791,373.492,175.489,41.037,158.034
C01317=1055.410,426.546,373.541,175.480,41.027,158.031
C01318=1055.400,426.301,373.588,175.469,41.017,158.028
C01319=1055.391,426.056,373.635,175.459,41.007,158.024
C01320=1055.381,425.811,373.682,175.450,40.997,158.021
C01321=1055.371,425.565,373.730,175.440,40.987,158.018
C01322=1055.361,425.320,373.777,175.430,40.977,158.015
C01323=1055.351,425.074,373.825,175.420,40.967,158.012
C01324=1055.341,424.829,373.873,175.411,40.957,158.009
C01325=1055.331,424.583,373.920,175.402,40.947,158.006
C01326=1055.322,424.339,373.967,175.392,40.937,158.002
C01327=1055.312,424.093,374.014,175.382,40.928,157.999
C01328=1055.303,423.848,374.062,175.372,40.918,157.996
C01329=1055.293,423.603,374.108,175.363,40.908,157.993
C01330=1055.283,423.357,374.156,175.353,40.899,157.990
C01331=1055.274,423.112,374.203,175.344,40.888,157.987
C01332=1055.264,422.866,374.250,175.335,40.879,157.984
C01333=1055.254,422.621,374.297,175.325,40.869,157.981
C01334=1055.245,422.376,374.345,175.316,40.860,157.978
C01335=1055.235,422.130,374.391,175.307,40.850,157.975
C01336=1055.226,421.884,374.438,175.297,40.840,157.972
C01337=1055.217,421.640,374.485,175.288,40.831,157.969
C01338=1055.207,421.394,374.531,175.279,40.821,157.966
C01339=1055.198,421.149,374.579,175.270,40.812,157.963
C01340=1055.188,420.903,374.625,175.260,40.803,157.960
C01341=1055.179,420.658,374.671,175.251,40.793,157.958
C01342=1055.170,420.412,374.718,175.242,40.784,157.955
C01343=1055.160,420.167,374.765,175.233,40.774,157.952
C01344=1055.151,419.922,374.811,175.224,40.765,157.949
C01345=1055.142,419.676,374.857,175.214,40.756,157.946
C01346=1055.132,419.430,374.905,175.206,40.746,157.943
C01347=1055.123,419.185,374.951,175.197,40.737,157.940
C01348=1055.113,418.939,374.997,175.188,40.728,157.938
C01349=1055.104,418.693,375.043,175.179,40.719,157.935
C01350=1055.095,418.448,375.089,175.170,40.709,157.932
C01351=1055.085,418.202,375.135,175.162,40.700,157.929
C01352=1055.076,417.957,375.181,175.153,40.692,157.926
C01353=1055.067,417.712,375.227,175.144,40.682,157.923
C01354=1055.053,417.355,375.294,175.131,40.669,157.919
C01355=1055.040,416.998,375.361,175.118,40.656,157.915
C01356=1055.026,416.642,375.427,175.106,40.643,157.911
C01357=1055.013,416.285,375.494,175.093,40.630,157.907
C01358=1055.004,416.040,375.539,175.084,40.621,157.905
C01359=1054.994,415.794,375.586,175.077,40.612,157.902
C01360=1054.985,415.548,375.631,175.068,40.603,157.899
C01361=1054.976,415.302,375.678,175.059,40.594,157.897
C01362=1054.967,415.057,375.723,175.051,40.586,157.894
C01363=1054.958,414.811,375.769,175.042,40.577,157.891
C01364=1054.949,414.565,375.814,175.034,40.568,157.889
C01365=1054.940,414.320,375.860,175.025,40.559,157.886
C01366=1054.930,414.074,375.905,175.017,40.550,157.883
C01367=1054.921,413.828,375.950,175.008,40.542,157.881
C01368=1054.913,413.583,375.995,175.001,40.533,157.878
C01369=1054.904,413.337,376.041,174.992,40.524,157.875
C01370=1054.895,413.092,376.086,174.984,40.515,157.873
C01371=1054.886,412.846,376.132,174.975,40.507,157.870
C01372=1054.876,412.600,376.177,174.967,40.499,157.868
C01373=1054.867,412.354,376.222,174.959,40.490,157.865
C01374=1054.859,412.108,376.267,174.951,40.482,157.863
C01375=1054.849,411.863,376.311,174.942,40.473,157.860
C01376=1054.840,411.617,376.357,174.935,40.465,157.858
C01377=1054.831,411.371,376.402,174.926,40.456,157.855
C01378=1054.823,411.125,376.447,174.918,40.448,157.853
C01379=1054.813,410.880,376.491,174.910,40.439,157.850
C01380=1054.804,410.634,376.537,174.902,40.431,157.847
C01381=1054.795,410.388,376.581,174.894,40.423,157.845
C01382=1054.787,410.143,376.626,174.886,40.414,157.843
C01383=1054.778,409.896,376.671,174.878,40.406,157.840
C01384=1054.768,409.651,376.716,174.870,40.397,157.837
C01385=1054.760,409.405,376.760,174.862,40.389,157.835
C01386=1054.751,409.158,376.805,174.854,40.381,157.833
C01387=1054.742,408.913,376.849,174.846,40.373,157.830
C01388=1054.734,408.667,376.894,174.839,40.364,157.828
C01389=1054.725,408.421,376.938,174.831,40.357,157.825
C01390=1054.716,408.176,376.983,174.823,40.349,157.823
C01391=1054.707,407.929,377.028,174.815,40.340,157.820
C01392=1054.698,407.684,377.071,174.807,40.332,157.818
C01393=1054.690,407.438,377.116,174.800,40.324,157.816
C01394=1054.682,407.192,377.160,174.792,40.316,157.813
C01395=1054.672,406.946,377.205,174.784,40.308,157.811
C01396=1054.664,406.701,377.250,174.776,40.300,157.809
C01397=1054.654,406.454,377.294,174.769,40.292,157.806
C01398=1054.641,406.071,377.363,174.757,40.279,157.802
C01399=1054.628,405.689,377.431,174.745,40.267,157.799
C01400=1054.615,405.306,377.500,174.733,40.254,157.795
C01401=1054.601,404.923,377.569,174.721,40.242,157.791
C01402=1054.593,404.677,377.612,174.714,40.234,157.789
C01403=1054.584,404.430,377.657,174.707,40.226,157.787
C01404=1054.575,404.185,377.700,174.699,40.219,157.785
C01405=1054.568,403.938,377.744,174.692,40.211,157.782
C01406=1054.559,403.708,377.785,174.685,40.204,157.780
C01407=1054.551,403.478,377.826,174.678,40.196,157.778
C01408=1054.544,403.249,377.867,174.671,40.189,157.776
C01409=1054.536,403.019,377.907,174.664,40.182,157.774
C01410=1054.527,402.790,377.948,174.658,40.175,157.772
C01411=1054.519,402.560,377.989,174.651,40.168,157.770
C01412=1054.511,402.330,378.030,174.644,40.161,157.768
C01413=1054.503,402.100,378.071,174.637,40.153,157.766
C01414=1054.494,401.854,378.114,174.630,40.146,157.763
C01415=1054.486,401.608,378.158,174.623,40.138,157.761
C01416=1054.478,401.362,378.201,174.615,40.130,157.759
C01417=1054.469,401.116,378.244,174.608,40.123,157.757
C01418=1054.461,400.870,378.287,174.601,40.115,157.754
C01419=1054.452,400.625,378.331,174.594,40.108,157.752
C01420=1054.444,400.378,378.374,174.586,40.101,157.750
C01421=1054.434,400.132,378.417,174.579,40.093,157.748
C01422=1054.427,399.885,378.461,174.572,40.086,157.746
C01423=1054.418,399.639,378.504,174.566,40.078,157.744
C01424=1054.410,399.393,378.547,174.559,40.071,157.742
C01425=1054.401,399.147,378.590,174.551,40.063,157.739
C01426=1054.393,398.901,378.633,174.544,40.056,157.737
C01427=1054.384,398.655,378.676,174.537,40.049,157.735
C01428=1054.376,398.410,378.719,174.530,40.041,157.733
C01429=1054.368,398.164,378.762,174.524,40.034,157.731
C01430=1054.359,397.918,378.805,174.516,40.027,157.729
C01431=1054.352,397.671,378.848,174.509,40.019,157.727
C01432=1054.343,397.425,378.891,174.502,40.012,157.725
C01433=1054.335,397.179,378.934,174.495,40.005,157.723
C01434=1054.326,396.932,378.977,174.489,39.998,157.721
C01435=1054.318,396.686,379.019,174.482,39.991,157.718
C01436=1054.310,396.440,379.062,174.475,39.983,157.716
C01437=1054.302,396.194,379.105,174.467,39.976,157.714
C01438=1054.293,395.948,379.147,174.461,39.969,157.712
C01439=1054.284,395.702,379.189,174.454,39.962,157.710
C01440=1054.276,395.455,379.232,174.447,39.955,157.708
C01441=1054.268,395.210,379.274,174.440,39.948,157.706
C01442=1054.260,394.963,379.317,174.434,39.941,157.704
C01443=1054.251,394.717,379.360,174.427,39.934,157.702
C01444=1054.244,394.471,379.402,174.420,39.927,157.700
C01445=1054.235,394.225,379.445,174.414,39.919,157.698
C01446=1054.227,393.978,379.487,174.407,39.913,157.696
C01447=1054.219,393.733,379.528,174.400,39.906,157.694
C01448=1054.211,393.486,379.571,174.394,39.898,157.692
C01449=1054.202,393.240,379.614,174.387,39.892,157.690
C01450=1054.195,392.994,379.656,174.380,39.885,157.688
C01451=1054.186,392.747,379.698,174.374,39.878,157.686
C01452=1054.179,392.501,379.740,174.367,39.871,157.684
C01453=1054.170,392.255,379.782,174.361,39.864,157.682
C01454=1054.161,392.009,379.825,174.354,39.857,157.680
C01455=1054.154,391.763,379.867,174.347,39.851,157.678
C01456=1054.145,391.517,379.908,174.341,39.844,157.677
C01457=1054.137,391.271,379.950,174.334,39.837,157.675
C01458=1054.129,391.024,379.993,174.328,39.830,157.673
C01459=1054.121,390.778,380.033,174.321,39.823,157.671
C01460=1054.113,390.531,380.075,174.314,39.816,157.669
C01461=1054.105,390.285,380.117,174.308,39.810,157.667
C01462=1054.097,390.039,380.159,174.302,39.803,157.665
C01463=1054.089,389.793,380.201,174.296,39.796,157.663
C01464=1054.081,389.547,380.243,174.289,39.790,157.661
C01465=1054.072,389.300,380.285,174.283,39.783,157.659
C01466=1054.062,388.967,380.341,174.274,39.774,157.657
C01467=1054.051,388.635,380.397,174.266,39.765,157.654
C01468=1054.039,388.302,380.453,174.257,39.756,157.652
C01469=1054.029,387.970,380.508,174.248,39.747,157.649
C01470=1054.021,387.723,380.550,174.242,39.741,157.648
C01471=1054.013,387.477,380.591,174.236,39.734,157.646
C01472=1054.004,387.230,380.633,174.229,39.728,157.644
C01473=1053.996,386.984,380.674,174.224,39.721,157.642
C01474=1053.988,386.738,380.715,174.217,39.715,157.640
C01475=1053.981,386.492,380.756,174.211,39.708,157.638
C01476=1053.972,386.245,380.798,174.204,39.702,157.637
C01477=1053.964,385.999,380.839,174.198,39.696,157.635
C01478=1053.957,385.752,380.880,174.193,39.689,157.633
C01479=1053.948,385.507,380.921,174.186,39.683,157.631
C01480=1053.940,385.259,380.963,174.180,39.677,157.629
C01481=1053.932,385.013,381.004,174.173,39.670,157.628
C01482=1053.924,384.767,381.044,174.168,39.664,157.626
C01483=1053.917,384.520,381.086,174.162,39.657,157.624
C01484=1053.909,384.274,381.127,174.155,39.651,157.622
C01485=1053.901,384.027,381.168,174.149,39.645,157.621
C01486=1053.893,383.781,381.209,174.144,39.638,157.619
C01487=1053.885,383.535,381.250,174.137,39.632,157.617
C01488=1053.877,383.288,381.291,174.131,39.626,157.615
C01489=1053.869,383.042,381.332,174.125,39.619,157.614
C01490=1053.861,382.795,381.372,174.119,39.613,157.612
C01491=1053.854,382.549,381.413,174.113,39.607,157.610
C01492=1053.846,382.303,381.454,174.107,39.601,157.608
C01493=1053.838,382.056,381.495,174.101,39.594,157.607
C01494=1053.831,381.810,381.536,174.095,39.589,157.605
C01495=1053.823,381.563,381.576,174.089,39.582,157.603
C01496=1053.815,381.317,381.617,174.083,39.576,157.601
C01497=1053.808,381.070,381.658,174.077,39.570,157.600
C01498=1053.800,380.824,381.698,174.071,39.564,157.598
C01499=1053.792,380.577,381.739,174.065,39.557,157.596
C01500=1053.785,380.330,381.780,174.060,39.551,157.595
C01501=1053.777,380.084,381.820,174.054,39.545,157.593
C01502=1053.769,379.838,381.861,174.048,39.539,157.591
C01503=1053.761,379.591,381.901,174.042,39.533,157.590
C01504=1053.753,379.344,381.941,174.036,39.527,157.588
C01505=1053.745,379.097,381.981,174.031,39.521,157.586
C01506=1053.737,378.851,382.022,174.024,39.515,157.585
C01507=1053.729,378.604,382.062,174.019,39.509,157.583
C01508=1053.721,378.358,382.102,174.013,39.503,157.581
C01509=1053.714,378.111,382.142,174.007,39.497,157.580
C01510=1053.706,377.865,382.183,174.002,39.491,157.578
C01511=1053.699,377.619,382.223,173.995,39.485,157.577
C01512=1053.691,377.372,382.262,173.990,39.479,157.575
C01513=1053.683,377.125,382.303,173.984,39.474,157.573
C01514=1053.675,376.879,382.343,173.978,39.468,157.572
C01515=1053.667,376.632,382.383,173.973,39.462,157.570
C01516=1053.660,376.385,382.423,173.967,39.456,157.568
C01517=1053.652,376.139,382.463,173.962,39.450,157.567
C01518=1053.644,375.892,382.503,173.956,39.444,157.565
C01519=1053.637,375.645,382.543,173.950,39.438,157.564
C01520=1053.629,375.398,382.583,173.944,39.432,157.562
C01521=1053.622,375.152,382.622,173.939,39.427,157.560
C01522=1053.612,374.851,382.671,173.932,39.420,157.559
C01523=1053.603,374.551,382.720,173.925,39.413,157.557
C01524=1053.594,374.250,382.768,173.918,39.406,157.555
C01525=1053.584,373.949,382.817,173.911,39.399,157.553
C01526=1053.577,373.703,382.857,173.906,39.393,157.551
C01527=1053.570,373.456,382.897,173.900,39.387,157.550
C01528=1053.562,373.209,382.937,173.895,39.382,157.548
C01529=1053.554,372.963,382.976,173.889,39.376,157.547
C01530=1053.546,372.716,383.015,173.884,39.370,157.545
C01531=1053.540,372.470,383.054,173.878,39.364,157.544
C01532=1053.532,372.223,383.094,173.873,39.359,157.542
C01533=1053.524,371.976,383.134,173.867,39.353,157.540
C01534=1053.517,371.730,383.174,173.862,39.347,157.539
C01535=1053.510,371.482,383.213,173.856,39.342,157.537
C01536=1053.501,371.236,383.252,173.851,39.336,157.536
C01537=1053.494,370.989,383.292,173.846,39.331,157.534
C01538=1053.487,370.742,383.331,173.840,39.325,157.533
C01539=1053.479,370.496,383.370,173.835,39.319,157.531
C01540=1053.471,370.248,383.409,173.829,39.314,157.530
C01541=1053.464,370.002,383.449,173.824,39.309,157.528
C01542=1053.456,369.756,383.488,173.818,39.303,157.527
C01543=1053.448,369.508,383.527,173.813,39.297,157.525
C01544=1053.440,369.262,383.566,173.808,39.292,157.524
C01545=1053.433,369.015,383.605,173.802,39.287,157.522
C01546=1053.426,368.768,383.644,173.797,39.281,157.521
C01547=1053.418,368.521,383.684,173.791,39.275,157.519
C01548=1053.411,368.274,383.722,173.787,39.270,157.518
C01549=1053.403,368.028,383.761,173.782,39.265,157.517
C01550=1053.396,367.781,383.801,173.776,39.259,157.515
C01551=1053.389,367.534,383.839,173.771,39.254,157.514
C01552=1053.381,367.287,383.878,173.765,39.248,157.512
C01553=1053.374,367.041,383.918,173.760,39.243,157.511
C01554=1053.365,366.794,383.956,173.755,39.238,157.509
C01555=1053.359,366.547,383.995,173.749,39.232,157.508
C01556=1053.352,366.300,384.034,173.744,39.227,157.506
C01557=1053.344,366.053,384.072,173.740,39.221,157.505
C01558=1053.337,365.806,384.112,173.734,39.216,157.504
C01559=1053.329,365.560,384.150,173.729,39.211,157.502
C01560=1053.322,365.312,384.189,173.724,39.205,157.501
C01561=1053.314,365.066,384.228,173.718,39.200,157.499
C01562=1053.307,364.819,384.266,173.713,39.195,157.498
C01563=1053.300,364.573,384.305,173.708,39.190,157.496
C01564=1053.292,364.325,384.344,173.703,39.184,157.495
C01565=1053.285,364.078,384.383,173.698,39.179,157.494
C01566=1053.278,363.832,384.421,173.693,39.174,157.492
C01567=1053.271,363.585,384.460,173.687,39.169,157.491
C01568=1053.263,363.338,384.498,173.682,39.163,157.489
C01569=1053.255,363.091,384.537,173.678,39.158,157.488
C01570=1053.249,362.844,384.575,173.672,39.153,157.487
C01571=1053.241,362.597,384.613,173.667,39.147,157.485
C01572=1053.233,362.350,384.652,173.662,39.143,157.484
C01573=1053.226,362.103,384.691,173.657,39.137,157.482
C01574=1053.219,361.856,384.728,173.652,39.132,157.481
C01575=1053.212,361.609,384.766,173.647,39.127,157.480
C01576=1053.204,361.362,384.805,173.642,39.122,157.478
C01577=1053.197,361.115,384.843,173.636,39.117,157.477
C01578=1053.189,360.833,384.887,173.631,39.111,157.476
C01579=1053.180,360.552,384.930,173.626,39.105,157.474
C01580=1053.172,360.270,384.974,173.620,39.099,157.472
C01581=1053.164,359.988,385.018,173.614,39.093,157.471
C01582=1053.156,359.741,385.056,173.610,39.088,157.470
C01583=1053.149,359.494,385.093,173.604,39.084,157.468
C01584=1053.141,359.248,385.132,173.599,39.079,157.467
C01585=1053.134,359.001,385.169,173.594,39.073,157.466
C01586=1053.128,358.753,385.207,173.590,39.068,157.464
C01587=1053.120,358.507,385.245,173.584,39.064,157.463
C01588=1053.113,358.260,385.283,173.579,39.059,157.462
C01589=1053.105,358.012,385.322,173.575,39.053,157.460
C01590=1053.098,357.765,385.360,173.570,39.048,157.459
C01591=1053.091,357.518,385.397,173.565,39.044,157.458
C01592=1053.083,357.271,385.435,173.560,39.039,157.456
C01593=1053.076,357.024,385.473,173.555,39.034,157.455
C01594=1053.069,356.777,385.511,173.550,39.029,157.454
C01595=1053.062,356.530,385.548,173.546,39.024,157.453
C01596=1053.054,356.283,385.586,173.541,39.019,157.451
C01597=1053.047,356.036,385.624,173.535,39.014,157.450
C01598=1053.040,355.789,385.661,173.531,39.009,157.449
C01599=1053.032,355.542,385.699,173.526,39.004,157.447
C01600=1053.025,355.295,385.736,173.521,39.000,157.446
C01601=1053.018,355.048,385.774,173.517,38.995,157.445
C01602=1053.011,354.801,385.811,173.512,38.990,157.444
C01603=1053.003,354.553,385.849,173.507,38.985,157.442
C01604=1052.997,354.307,385.886,173.502,38.980,157.441
C01605=1052.989,354.060,385.924,173.497,38.975,157.440
C01606=1052.982,353.813,385.961,173.493,38.970,157.438
C01607=1052.975,353.566,385.999,173.488,38.966,157.437
C01608=1052.968,353.318,386.036,173.484,38.961,157.436
C01609=1052.960,353.071,386.074,173.478,38.956,157.435
C01610=1052.953,352.824,386.111,173.473,38.951,157.433
C01611=1052.946,352.577,386.149,173.469,38.946,157.432
C01612=1052.940,352.330,386.185,173.464,38.942,157.431
C01613=1052.932,352.083,386.223,173.460,38.937,157.430
C01614=1052.925,351.836,386.260,173.455,38.932,157.428
C01615=1052.918,351.589,386.298,173.451,38.927,157.427
C01616=1052.911,351.341,386.335,173.446,38.923,157.426
C01617=1052.904,351.095,386.371,173.441,38.918,157.425
C01618=1052.896,350.848,386.409,173.436,38.913,157.423
C01619=1052.889,350.600,386.446,173.432,38.908,157.422
C01620=1052.882,350.353,386.483,173.427,38.904,157.421
C01621=1052.875,350.105,386.521,173.422,38.899,157.420
C01622=1052.868,349.859,386.556,173.418,38.894,157.419
C01623=1052.861,349.612,386.594,173.413,38.890,157.417
C01624=1052.854,349.364,386.631,173.409,38.885,157.416
C01625=1052.846,349.117,386.668,173.404,38.881,157.415
C01626=1052.839,348.870,386.704,173.399,38.876,157.414
C01627=1052.832,348.623,386.742,173.394,38.871,157.413
C01628=1052.825,348.375,386.779,173.390,38.866,157.411
C01629=1052.819,348.129,386.816,173.385,38.862,157.410
C01630=1052.811,347.881,386.852,173.381,38.857,157.409
C01631=1052.804,347.634,386.889,173.377,38.853,157.408
C01632=1052.797,347.386,386.926,173.372,38.848,157.407
C01633=1052.790,347.140,386.962,173.368,38.843,157.405
C01634=1052.781,346.863,387.004,173.363,38.838,157.404
C01635=1052.773,346.586,387.045,173.358,38.834,157.403
C01636=1052.766,346.310,387.086,173.352,38.828,157.401
C01637=1052.758,346.033,387.127,173.347,38.823,157.400
C01638=1052.751,345.786,387.164,173.343,38.819,157.399
C01639=1052.744,345.539,387.200,173.338,38.814,157.398
C01640=1052.737,345.291,387.237,173.334,38.809,157.397
C01641=1052.730,345.044,387.273,173.329,38.805,157.396
C01642=1052.723,344.797,387.310,173.325,38.801,157.394
C01643=1052.716,344.549,387.346,173.321,38.796,157.393
C01644=1052.709,344.303,387.384,173.316,38.792,157.392
C01645=1052.701,344.055,387.420,173.312,38.787,157.391
C01646=1052.695,343.808,387.456,173.307,38.783,157.390
C01647=1052.687,343.561,387.492,173.303,38.778,157.389
C01648=1052.681,343.314,387.529,173.299,38.774,157.388
C01649=1052.673,343.066,387.565,173.294,38.769,157.386
C01650=1052.667,342.819,387.601,173.290,38.765,157.385
C01651=1052.659,342.572,387.638,173.286,38.761,157.384
C01652=1052.653,342.325,387.674,173.281,38.756,157.383
C01653=1052.645,342.077,387.710,173.277,38.752,157.382
C01654=1052.639,341.829,387.746,173.272,38.747,157.381
C01655=1052.632,341.582,387.782,173.268,38.743,157.380
C01656=1052.625,341.335,387.818,173.264,38.739,157.378
C01657=1052.618,341.087,387.855,173.259,38.734,157.377
C01658=1052.611,340.841,387.891,173.255,38.730,157.376
C01659=1052.603,340.593,387.927,173.251,38.725,157.375
C01660=1052.597,340.346,387.963,173.246,38.721,157.374
C01661=1052.589,340.098,387.999,173.242,38.717,157.373
C01662=1052.582,339.851,388.035,173.238,38.713,157.372
C01663=1052.576,339.604,388.071,173.233,38.708,157.371
C01664=1052.568,339.356,388.107,173.229,38.704,157.370
C01665=1052.561,339.110,388.143,173.225,38.699,157.369
C01666=1052.555,338.862,388.179,173.220,38.695,157.367
C01667=1052.548,338.614,388.215,173.216,38.691,157.366
C01668=1052.541,338.368,388.250,173.212,38.687,157.365
C01669=1052.534,338.119,388.287,173.208,38.682,157.364
C01670=1052.527,337.873,388.322,173.203,38.678,157.363
C01671=1052.520,337.626,388.358,173.199,38.674,157.362
C01672=1052.514,337.378,388.394,173.195,38.669,157.361
C01673=1052.506,337.131,388.430,173.190,38.665,157.360
C01674=1052.499,336.883,388.465,173.186,38.661,157.359
C01675=1052.493,336.636,388.502,173.182,38.656,157.358
C01676=1052.486,336.388,388.537,173.179,38.653,157.357
C01677=1052.479,336.141,388.572,173.174,38.648,157.355
C01678=1052.472,335.894,388.608,173.170,38.644,157.354
C01679=1052.464,335.646,388.644,173.166,38.640,157.353
C01680=1052.457,335.399,388.680,173.162,38.635,157.352
C01681=1052.451,335.152,388.715,173.157,38.632,157.351
C01682=1052.445,334.904,388.750,173.153,38.627,157.350
C01683=1052.437,334.656,388.786,173.149,38.623,157.349
C01684=1052.430,334.409,388.822,173.145,38.619,157.348
C01685=1052.423,334.162,388.857,173.141,38.615,157.347
C01686=1052.417,333.915,388.892,173.136,38.611,157.346
C01687=1052.409,333.667,388.928,173.132,38.607,157.345
C01688=1052.402,333.420,388.963,173.128,38.602,157.344
C01689=1052.395,333.173,388.999,173.125,38.598,157.343
C01690=1052.388,332.892,389.039,173.119,38.593,157.342
C01691=1052.380,332.611,389.079,173.114,38.589,157.341
C01692=1052.372,332.331,389.119,173.110,38.584,157.339
C01693=1052.364,332.049,389.159,173.105,38.580,157.338
C01694=1052.357,331.802,389.194,173.101,38.575,157.337
C01695=1052.350,331.555,389.230,173.098,38.571,157.336
C01696=1052.344,331.307,389.265,173.094,38.567,157.335
C01697=1052.337,331.060,389.300,173.090,38.563,157.334
C01698=1052.330,330.813,389.335,173.085,38.559,157.333
C01699=1052.323,330.565,389.370,173.081,38.555,157.332
C01700=1052.317,330.318,389.405,173.077,38.551,157.331
C01701=1052.310,330.071,389.440,173.073,38.547,157.330
C01702=1052.302,329.823,389.476,173.069,38.542,157.329
C01703=1052.296,329.575,389.510,173.065,38.539,157.328
C01704=1052.289,329.327,389.545,173.062,38.535,157.327
C01705=1052.282,329.080,389.580,173.057,38.531,157.326
C01706=1052.275,328.833,389.615,173.053,38.527,157.325
C01707=1052.268,328.585,389.650,173.049,38.523,157.324
C01708=1052.261,328.338,389.684,173.045,38.519,157.323
C01709=1052.254,328.090,389.719,173.041,38.515,157.322
C01710=1052.247,327.842,389.755,173.037,38.511,157.321
C01711=1052.240,327.595,389.789,173.034,38.507,157.320
C01712=1052.233,327.347,389.824,173.029,38.503,157.319
C01713=1052.226,327.100,389.859,173.025,38.499,157.318
C01714=1052.219,326.852,389.893,173.021,38.495,157.317
C01715=1052.212,326.605,389.928,173.017,38.491,157.316
C01716=1052.205,326.358,389.962,173.013,38.487,157.315
C01717=1052.198,326.110,389.997,173.010,38.484,157.314
C01718=1052.191,325.862,390.032,173.006,38.480,157.313
C01719=1052.184,325.615,390.066,173.002,38.476,157.312
C01720=1052.177,325.367,390.101,172.998,38.472,157.311
C01721=1052.171,325.120,390.136,172.994,38.468,157.310
C01722=1052.164,324.872,390.170,172.989,38.464,157.309
C01723=1052.157,324.625,390.205,172.986,38.460,157.308
C01724=1052.150,324.377,390.239,172.982,38.456,157.307
C01725=1052.143,324.129,390.273,172.978,38.452,157.306
C01726=1052.137,323.883,390.308,172.974,38.448,157.305
C01727=1052.130,323.635,390.342,172.970,38.445,157.304
C01728=1052.123,323.388,390.377,172.966,38.441,157.303
C01729=1052.116,323.140,390.411,172.963,38.437,157.302
C01730=1052.109,322.893,390.446,172.959,38.433,157.301
C01731=1052.103,322.645,390.480,172.955,38.429,157.301
C01732=1052.095,322.397,390.514,172.951,38.425,157.300
C01733=1052.089,322.150,390.549,172.947,38.421,157.299
C01734=1052.082,321.903,390.583,172.944,38.417,157.298
C01735=1052.075,321.655,390.617,172.940,38.414,157.297
C01736=1052.068,321.408,390.652,172.936,38.410,157.296
C01737=1052.062,321.160,390.686,172.932,38.406,157.295
C01738=1052.055,320.912,390.720,172.928,38.402,157.294
C01739=1052.048,320.665,390.754,172.925,38.398,157.293
C01740=1052.042,320.417,390.788,172.921,38.394,157.292
C01741=1052.034,320.170,390.823,172.917,38.390,157.291
C01742=1052.028,319.922,390.857,172.913,38.387,157.290
C01743=1052.021,319.674,390.891,172.909,38.383,157.289
C01744=1052.015,319.427,390.925,172.906,38.379,157.288
C01745=1052.008,319.179,390.959,172.902,38.375,157.287
C01746=1052.000,318.893,391.000,172.898,38.371,157.286
C01747=1051.993,318.607,391.039,172.893,38.366,157.285
C01748=1051.985,318.321,391.078,172.889,38.362,157.284
C01749=1051.978,318.035,391.117,172.884,38.358,157.283
C01750=1051.970,317.788,391.151,172.881,38.354,157.282
C01751=1051.965,317.541,391.185,172.878,38.350,157.281
C01752=1051.957,317.293,391.219,172.874,38.346,157.280
C01753=1051.951,317.045,391.253,172.870,38.342,157.279
C01754=1051.944,316.798,391.287,172.866,38.339,157.278
C01755=1051.938,316.550,391.321,172.862,38.335,157.277
C01756=1051.931,316.302,391.355,172.859,38.331,157.276
C01757=1051.925,316.055,391.389,172.855,38.327,157.275
C01758=1051.918,315.807,391.423,172.851,38.324,157.275
C01759=1051.912,315.560,391.457,172.847,38.320,157.274
C01760=1051.905,315.312,391.491,172.843,38.316,157.273
C01761=1051.899,315.064,391.524,172.841,38.313,157.272
C01762=1051.892,314.817,391.558,172.837,38.309,157.271
C01763=1051.885,314.569,391.593,172.833,38.305,157.270
C01764=1051.879,314.322,391.626,172.829,38.301,157.269
C01765=1051.872,314.074,391.660,172.826,38.297,157.268
C01766=1051.866,313.827,391.694,172.822,38.293,157.267
C01767=1051.859,313.579,391.727,172.818,38.290,157.266
C01768=1051.853,313.331,391.761,172.815,38.286,157.265
C01769=1051.846,313.084,391.795,172.812,38.282,157.264
C01770=1051.839,312.836,391.828,172.808,38.279,157.264
C01771=1051.832,312.588,391.861,172.804,38.275,157.263
C01772=1051.826,312.341,391.895,172.800,38.272,157.262
C01773=1051.819,312.093,391.928,172.797,38.268,157.261
C01774=1051.812,311.845,391.962,172.793,38.264,157.260
C01775=1051.805,311.598,391.995,172.789,38.261,157.259
C01776=1051.798,311.350,392.028,172.785,38.257,157.258
C01777=1051.792,311.103,392.061,172.783,38.254,157.257
C01778=1051.785,310.855,392.095,172.779,38.250,157.257
C01779=1051.778,310.607,392.128,172.775,38.246,157.256
C01780=1051.771,310.360,392.162,172.772,38.243,157.255
C01781=1051.765,310.112,392.194,172.768,38.239,157.254
C01782=1051.758,309.864,392.228,172.764,38.236,157.253
C01783=1051.751,309.617,392.261,172.760,38.232,157.252
C01784=1051.744,309.369,392.293,172.758,38.228,157.251
C01785=1051.737,309.122,392.327,172.754,38.225,157.251
C01786=1051.730,308.873,392.360,172.750,38.221,157.250
C01787=1051.724,308.627,392.393,172.747,38.218,157.249
C01788=1051.717,308.378,392.426,172.743,38.214,157.248
C01789=1051.710,308.131,392.459,172.739,38.211,157.247
C01790=1051.703,307.883,392.493,172.737,38.207,157.246
C01791=1051.697,307.635,392.526,172.733,38.203,157.245
C01792=1051.691,307.388,392.559,172.729,38.200,157.245
C01793=1051.683,307.140,392.591,172.725,38.197,157.244
C01794=1051.676,306.893,392.625,172.722,38.193,157.243
C01795=1051.669,306.644,392.658,172.719,38.189,157.242
C01796=1051.663,306.397,392.690,172.715,38.186,157.241
C01797=1051.657,306.149,392.723,172.712,38.183,157.240
C01798=1051.650,305.902,392.757,172.708,38.179,157.239
C01799=1051.643,305.654,392.790,172.704,38.175,157.239
C01800=1051.637,305.406,392.822,172.701,38.172,157.238
C01801=1051.629,305.158,392.855,172.698,38.168,157.237
C01802=1051.623,304.877,392.892,172.694,38.164,157.236
C01803=1051.615,304.595,392.930,172.690,38.160,157.235
C01804=1051.607,304.314,392.967,172.685,38.156,157.234
C01805=1051.600,304.032,393.004,172.682,38.152,157.233
C01806=1051.593,303.784,393.037,172.679,38.149,157.232
C01807=1051.586,303.536,393.070,172.675,38.145,157.231
C01808=1051.580,303.289,393.102,172.671,38.141,157.230
C01809=1051.574,303.041,393.135,172.668,38.138,157.230
